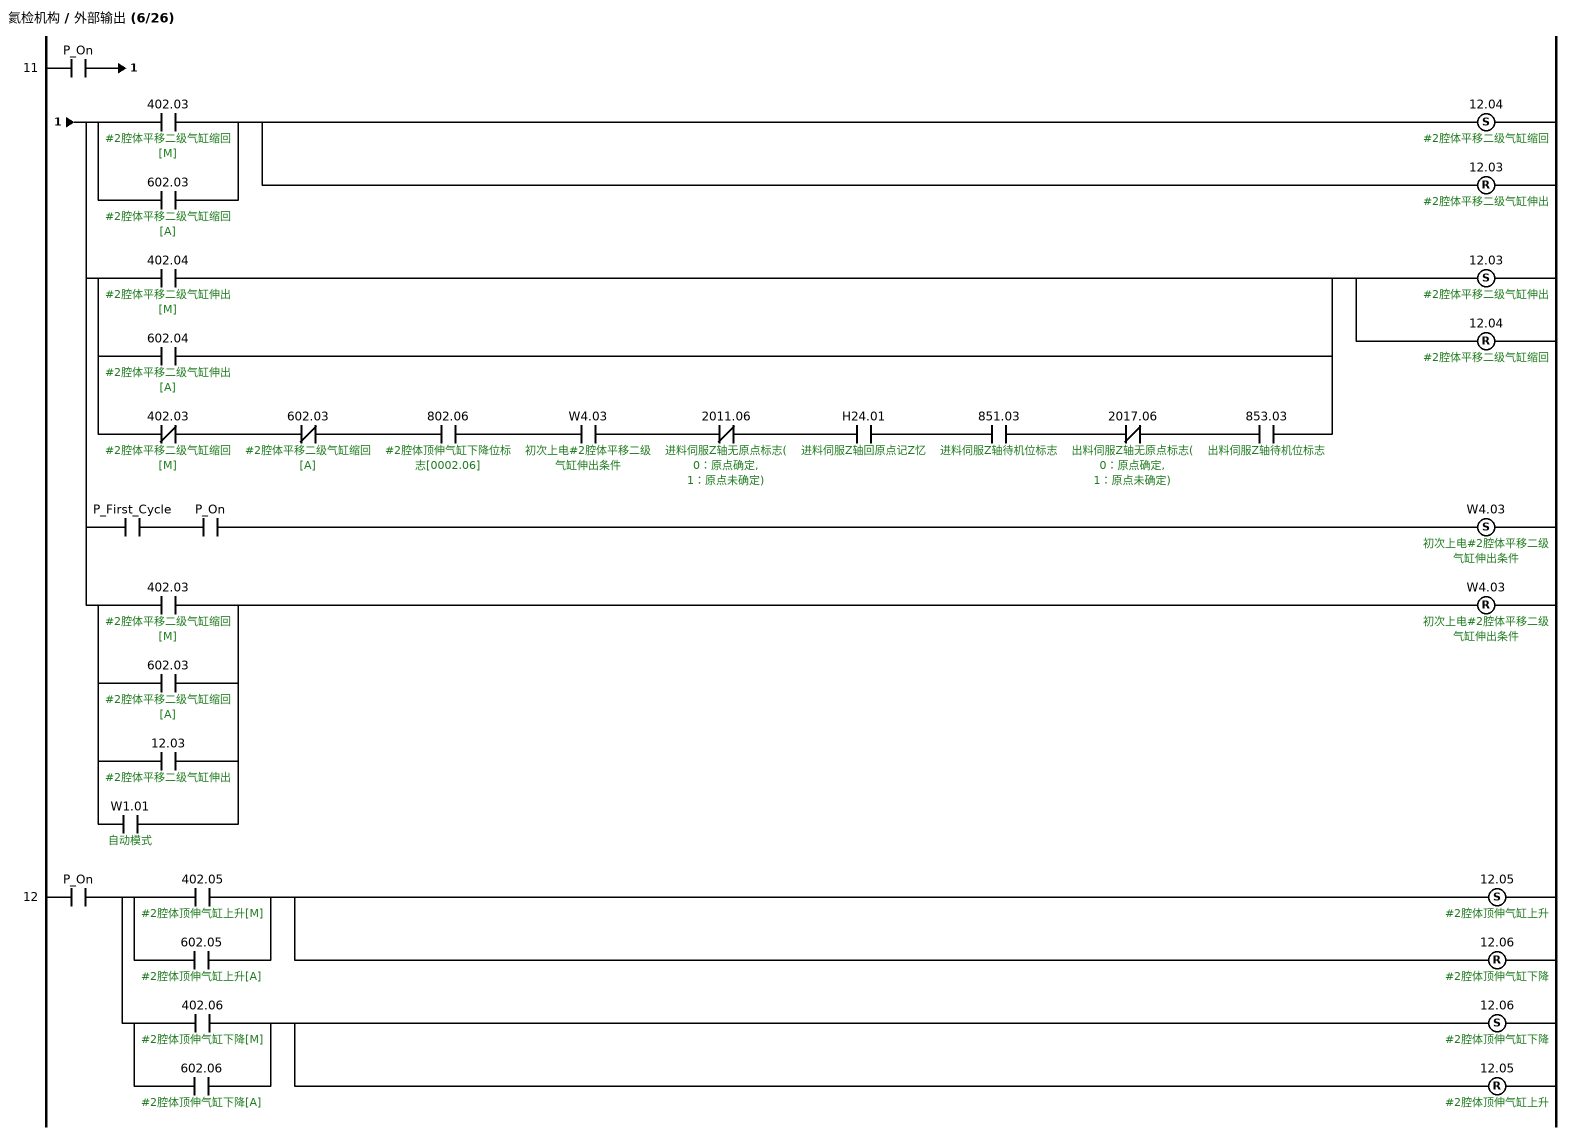
; [picture p432: 氦检机构 / 外部输出, rungs 11-12]
; rung 11
LD P_On
OUT TR0
LD 402.03  ; #2腔体平移二级气缸缩回[M]
OR 602.03  ; #2腔体平移二级气缸缩回[A]
ANDLD
SET 12.04  ; #2腔体平移二级气缸缩回
RSET 12.03  ; #2腔体平移二级气缸伸出
LD TR0
LD 402.04  ; #2腔体平移二级气缸伸出[M]
OR 602.04  ; #2腔体平移二级气缸伸出[A]
LDNOT 402.03  ; #2腔体平移二级气缸缩回[M]
ANDNOT 602.03  ; #2腔体平移二级气缸缩回[A]
AND 802.06  ; #2腔体顶伸气缸下降位标志[0002.06]
AND W4.03  ; 初次上电#2腔体平移二级气缸伸出条件
ANDNOT 2011.06  ; 进料伺服Z轴无原点标志(0：原点确定,1：原点未确定)
AND H24.01  ; 进料伺服Z轴回原点记Z忆
AND 851.03  ; 进料伺服Z轴待机位标志
ANDNOT 2017.06  ; 出料伺服Z轴无原点标志(0：原点确定,1：原点未确定)
AND 853.03  ; 出料伺服Z轴待机位标志
ORLD
ANDLD
SET 12.03  ; #2腔体平移二级气缸伸出
RSET 12.04  ; #2腔体平移二级气缸缩回
LD TR0
AND P_First_Cycle
AND P_On
SET W4.03  ; 初次上电#2腔体平移二级气缸伸出条件
LD TR0
LD 402.03  ; #2腔体平移二级气缸缩回[M]
OR 602.03  ; #2腔体平移二级气缸缩回[A]
OR 12.03  ; #2腔体平移二级气缸伸出
OR W1.01  ; 自动模式
ANDLD
RSET W4.03  ; 初次上电#2腔体平移二级气缸伸出条件
; rung 12
LD P_On
OUT TR0
LD 402.05  ; #2腔体顶伸气缸上升[M]
OR 602.05  ; #2腔体顶伸气缸上升[A]
ANDLD
SET 12.05  ; #2腔体顶伸气缸上升
RSET 12.06  ; #2腔体顶伸气缸下降
LD TR0
LD 402.06  ; #2腔体顶伸气缸下降[M]
OR 602.06  ; #2腔体顶伸气缸下降[A]
ANDLD
SET 12.06  ; #2腔体顶伸气缸下降
RSET 12.05  ; #2腔体顶伸气缸上升

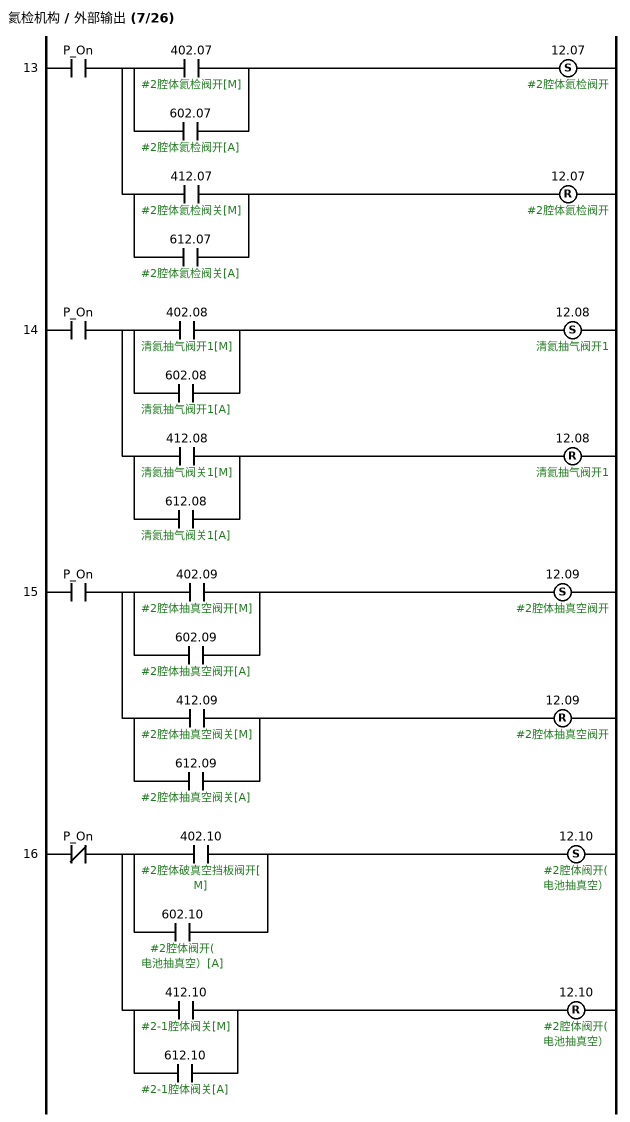
; rung 13
LD P_On
OUT TR0
LD 402.07  ; #2腔体氦检阀开[M]
OR 602.07  ; #2腔体氦检阀开[A]
ANDLD
SET 12.07  ; #2腔体氦检阀开
LD TR0
LD 412.07  ; #2腔体氦检阀关[M]
OR 612.07  ; #2腔体氦检阀关[A]
ANDLD
RSET 12.07  ; #2腔体氦检阀开
; rung 14
LD P_On
OUT TR0
LD 402.08  ; 清氦抽气阀开1[M]
OR 602.08  ; 清氦抽气阀开1[A]
ANDLD
SET 12.08  ; 清氦抽气阀开1
LD TR0
LD 412.08  ; 清氦抽气阀关1[M]
OR 612.08  ; 清氦抽气阀关1[A]
ANDLD
RSET 12.08  ; 清氦抽气阀开1
; rung 15
LD P_On
OUT TR0
LD 402.09  ; #2腔体抽真空阀开[M]
OR 602.09  ; #2腔体抽真空阀开[A]
ANDLD
SET 12.09  ; #2腔体抽真空阀开
LD TR0
LD 412.09  ; #2腔体抽真空阀关[M]
OR 612.09  ; #2腔体抽真空阀关[A]
ANDLD
RSET 12.09  ; #2腔体抽真空阀开
; rung 16
LDNOT P_On
OUT TR0
LD 402.10  ; #2腔体破真空挡板阀开[M]
OR 602.10  ; #2腔体阀开(电池抽真空）[A]
ANDLD
SET 12.10  ; #2腔体阀开(电池抽真空）
LD TR0
LD 412.10  ; #2-1腔体阀关[M]
OR 612.10  ; #2-1腔体阀关[A]
ANDLD
RSET 12.10  ; #2腔体阀开(电池抽真空）

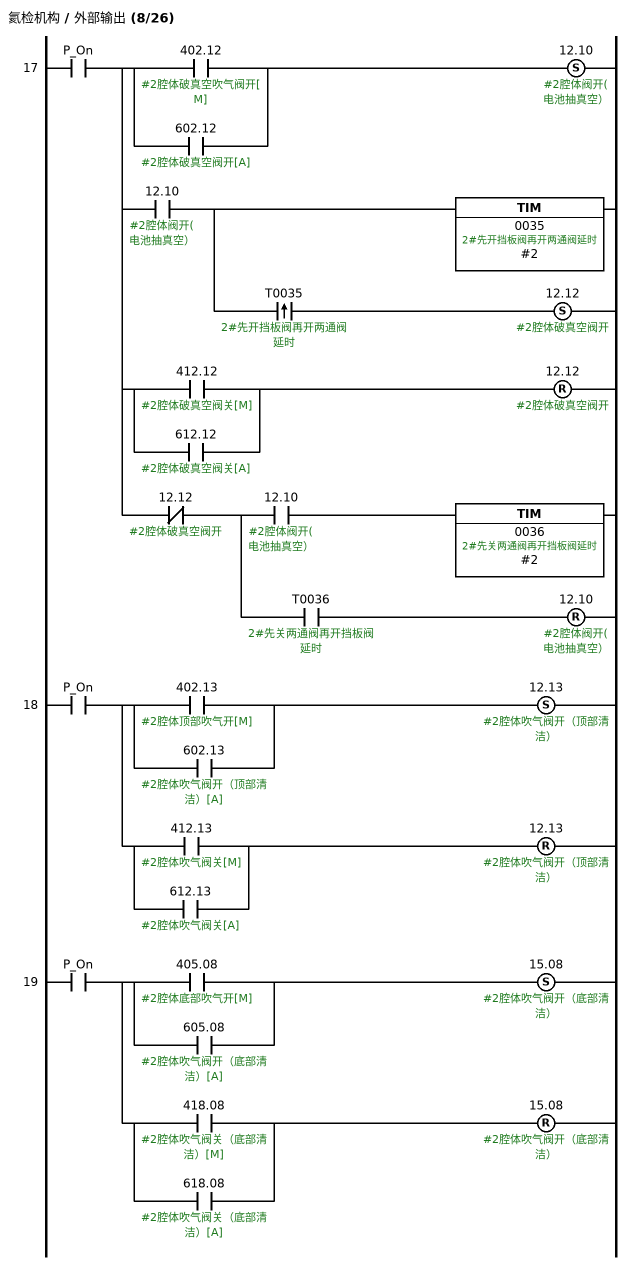
; rung 17
LD P_On
OUT TR0
LD 402.12  ; #2腔体破真空吹气阀开[M]
OR 602.12  ; #2腔体破真空阀开[A]
ANDLD
SET 12.10  ; #2腔体阀开(电池抽真空）
LD TR0
AND 12.10  ; #2腔体阀开(电池抽真空）
TIM 0035 #2  ; 2#先开挡板阀再开两通阀延时
@AND T0035  ; 2#先开挡板阀再开两通阀延时
SET 12.12  ; #2腔体破真空阀开
LD TR0
LD 412.12  ; #2腔体破真空阀关[M]
OR 612.12  ; #2腔体破真空阀关[A]
ANDLD
RSET 12.12  ; #2腔体破真空阀开
LD TR0
ANDNOT 12.12  ; #2腔体破真空阀开
OUT TR0
AND 12.10  ; #2腔体阀开(电池抽真空）
TIM 0036 #2  ; 2#先关两通阀再开挡板阀延时
LD TR0
AND T0036  ; 2#先关两通阀再开挡板阀延时
RSET 12.10  ; #2腔体阀开(电池抽真空）
; rung 18
LD P_On
OUT TR0
LD 402.13  ; #2腔体顶部吹气开[M]
OR 602.13  ; #2腔体吹气阀开（顶部清洁）[A]
ANDLD
SET 12.13  ; #2腔体吹气阀开（顶部清洁）
LD TR0
LD 412.13  ; #2腔体吹气阀关[M]
OR 612.13  ; #2腔体吹气阀关[A]
ANDLD
RSET 12.13  ; #2腔体吹气阀开（顶部清洁）
; rung 19
LD P_On
OUT TR0
LD 405.08  ; #2腔体底部吹气开[M]
OR 605.08  ; #2腔体吹气阀开（底部清洁）[A]
ANDLD
SET 15.08  ; #2腔体吹气阀开（底部清洁）
LD TR0
LD 418.08  ; #2腔体吹气阀关（底部清洁）[M]
OR 618.08  ; #2腔体吹气阀关（底部清洁）[A]
ANDLD
RSET 15.08  ; #2腔体吹气阀开（底部清洁）

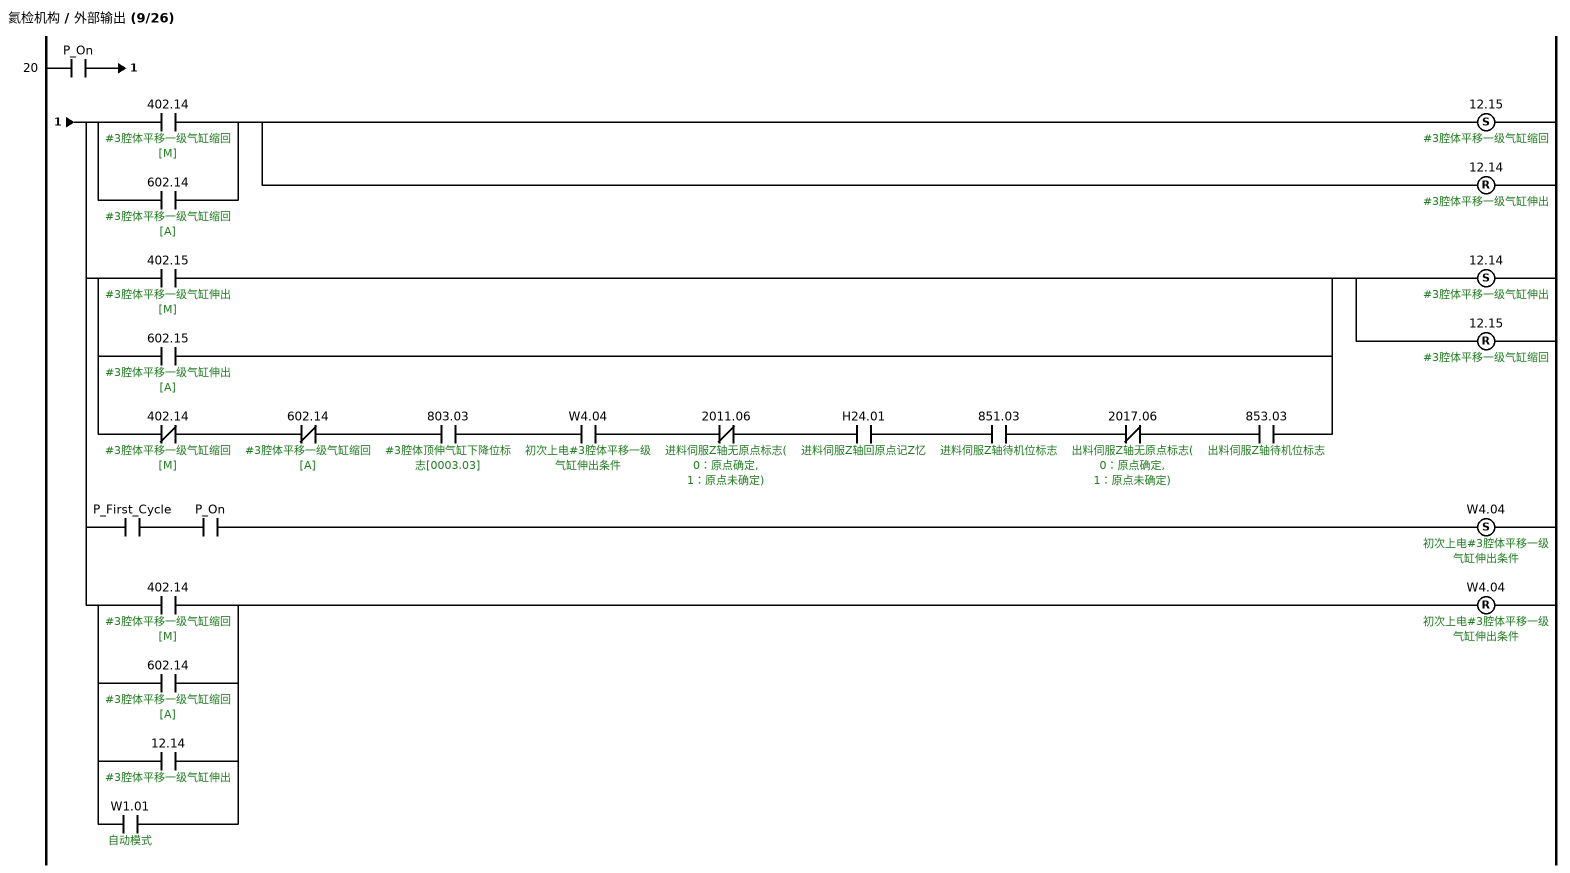
; rung 20
LD P_On
OUT TR0
LD 402.14  ; #3腔体平移一级气缸缩回[M]
OR 602.14  ; #3腔体平移一级气缸缩回[A]
ANDLD
SET 12.15  ; #3腔体平移一级气缸缩回
RSET 12.14  ; #3腔体平移一级气缸伸出
LD TR0
LD 402.15  ; #3腔体平移一级气缸伸出[M]
OR 602.15  ; #3腔体平移一级气缸伸出[A]
LDNOT 402.14  ; #3腔体平移一级气缸缩回[M]
ANDNOT 602.14  ; #3腔体平移一级气缸缩回[A]
AND 803.03  ; #3腔体顶伸气缸下降位标志[0003.03]
AND W4.04  ; 初次上电#3腔体平移一级气缸伸出条件
ANDNOT 2011.06  ; 进料伺服Z轴无原点标志(0：原点确定,1：原点未确定)
AND H24.01  ; 进料伺服Z轴回原点记Z忆
AND 851.03  ; 进料伺服Z轴待机位标志
ANDNOT 2017.06  ; 出料伺服Z轴无原点标志(0：原点确定,1：原点未确定)
AND 853.03  ; 出料伺服Z轴待机位标志
ORLD
ANDLD
SET 12.14  ; #3腔体平移一级气缸伸出
RSET 12.15  ; #3腔体平移一级气缸缩回
LD TR0
AND P_First_Cycle
AND P_On
SET W4.04  ; 初次上电#3腔体平移一级气缸伸出条件
LD TR0
LD 402.14  ; #3腔体平移一级气缸缩回[M]
OR 602.14  ; #3腔体平移一级气缸缩回[A]
OR 12.14  ; #3腔体平移一级气缸伸出
OR W1.01  ; 自动模式
ANDLD
RSET W4.04  ; 初次上电#3腔体平移一级气缸伸出条件

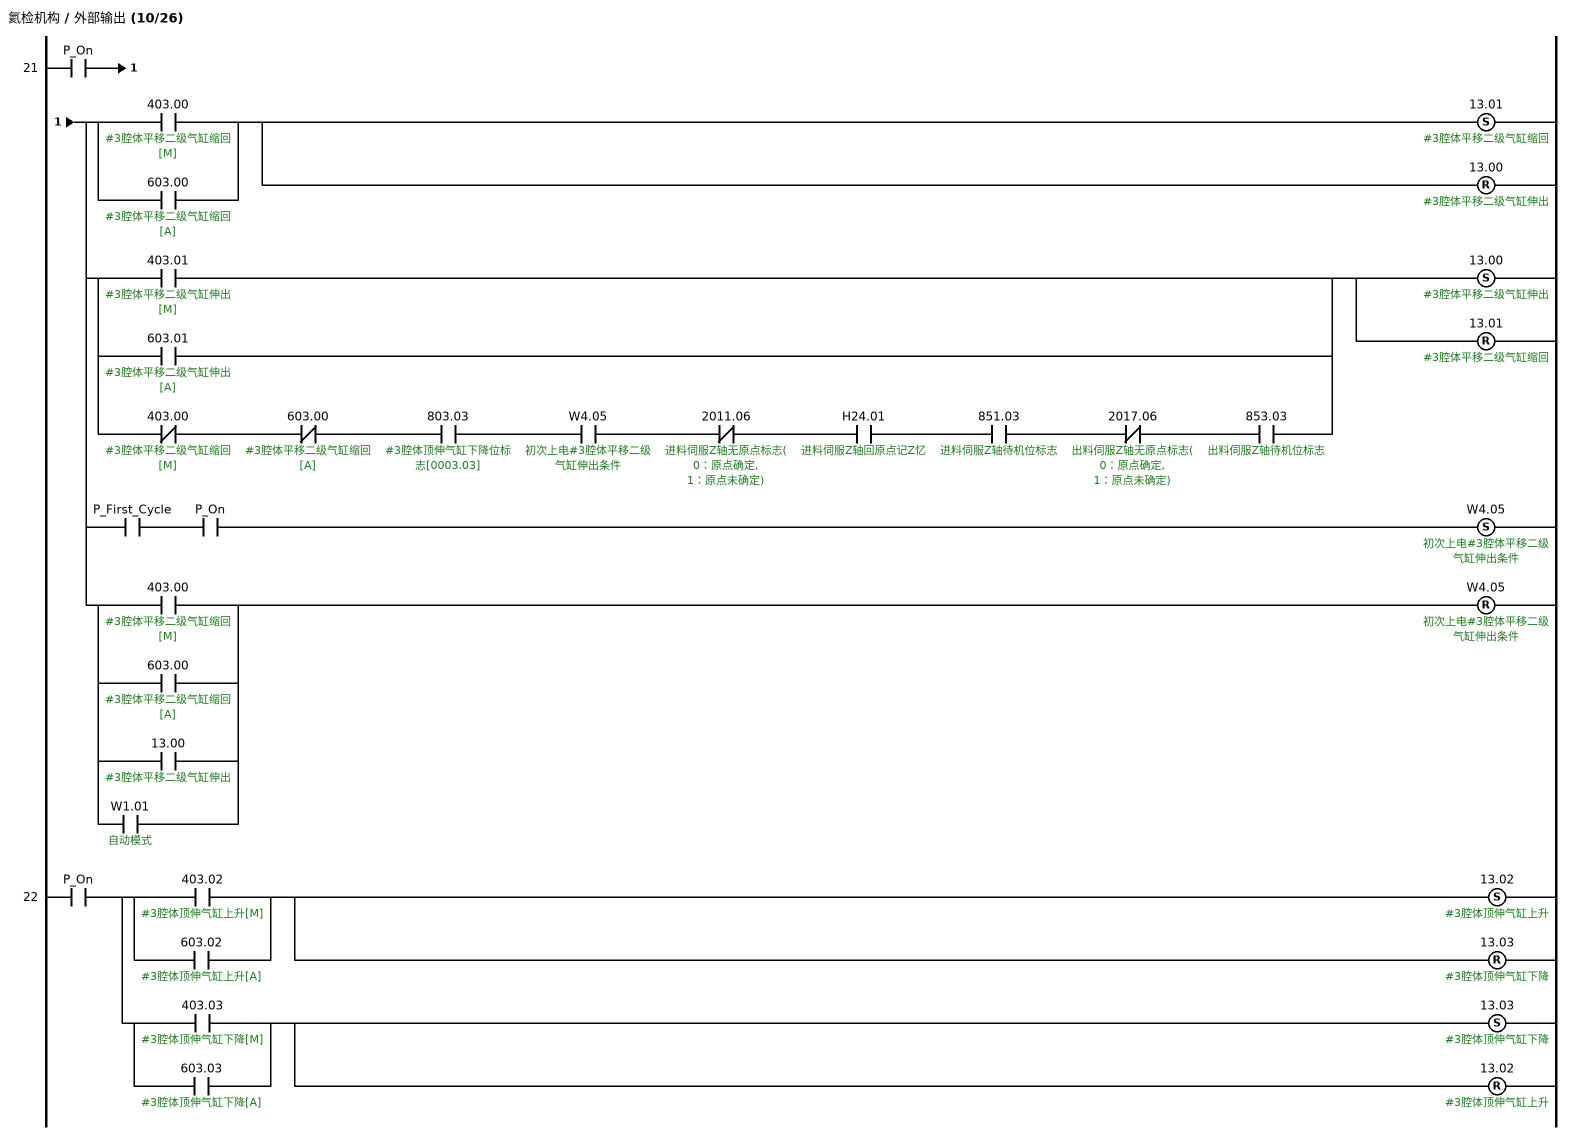
; rung 21
LD P_On
OUT TR0
LD 403.00  ; #3腔体平移二级气缸缩回[M]
OR 603.00  ; #3腔体平移二级气缸缩回[A]
ANDLD
SET 13.01  ; #3腔体平移二级气缸缩回
RSET 13.00  ; #3腔体平移二级气缸伸出
LD TR0
LD 403.01  ; #3腔体平移二级气缸伸出[M]
OR 603.01  ; #3腔体平移二级气缸伸出[A]
LDNOT 403.00  ; #3腔体平移二级气缸缩回[M]
ANDNOT 603.00  ; #3腔体平移二级气缸缩回[A]
AND 803.03  ; #3腔体顶伸气缸下降位标志[0003.03]
AND W4.05  ; 初次上电#3腔体平移二级气缸伸出条件
ANDNOT 2011.06  ; 进料伺服Z轴无原点标志(0：原点确定,1：原点未确定)
AND H24.01  ; 进料伺服Z轴回原点记Z忆
AND 851.03  ; 进料伺服Z轴待机位标志
ANDNOT 2017.06  ; 出料伺服Z轴无原点标志(0：原点确定,1：原点未确定)
AND 853.03  ; 出料伺服Z轴待机位标志
ORLD
ANDLD
SET 13.00  ; #3腔体平移二级气缸伸出
RSET 13.01  ; #3腔体平移二级气缸缩回
LD TR0
AND P_First_Cycle
AND P_On
SET W4.05  ; 初次上电#3腔体平移二级气缸伸出条件
LD TR0
LD 403.00  ; #3腔体平移二级气缸缩回[M]
OR 603.00  ; #3腔体平移二级气缸缩回[A]
OR 13.00  ; #3腔体平移二级气缸伸出
OR W1.01  ; 自动模式
ANDLD
RSET W4.05  ; 初次上电#3腔体平移二级气缸伸出条件
; rung 22
LD P_On
OUT TR0
LD 403.02  ; #3腔体顶伸气缸上升[M]
OR 603.02  ; #3腔体顶伸气缸上升[A]
ANDLD
SET 13.02  ; #3腔体顶伸气缸上升
RSET 13.03  ; #3腔体顶伸气缸下降
LD TR0
LD 403.03  ; #3腔体顶伸气缸下降[M]
OR 603.03  ; #3腔体顶伸气缸下降[A]
ANDLD
SET 13.03  ; #3腔体顶伸气缸下降
RSET 13.02  ; #3腔体顶伸气缸上升

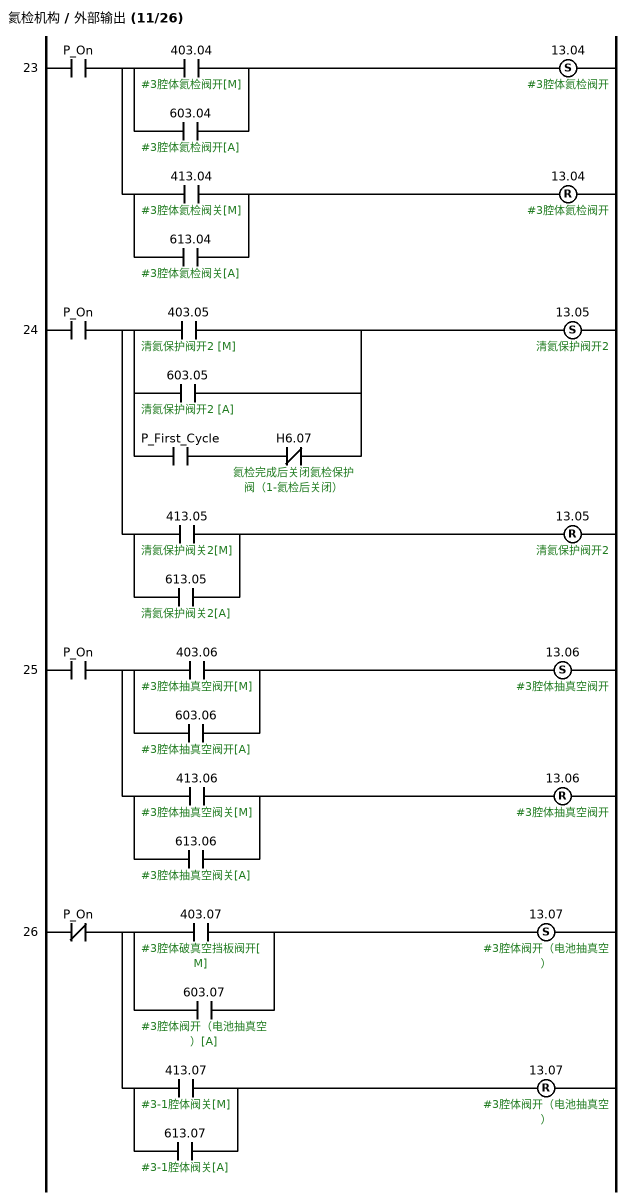
; rung 23
LD P_On
OUT TR0
LD 403.04  ; #3腔体氦检阀开[M]
OR 603.04  ; #3腔体氦检阀开[A]
ANDLD
SET 13.04  ; #3腔体氦检阀开
LD TR0
LD 413.04  ; #3腔体氦检阀关[M]
OR 613.04  ; #3腔体氦检阀关[A]
ANDLD
RSET 13.04  ; #3腔体氦检阀开
; rung 24
LD P_On
OUT TR0
LD 403.05  ; 清氦保护阀开2 [M]
OR 603.05  ; 清氦保护阀开2 [A]
LD P_First_Cycle  // 保证氦检仪开启时能将管路抽成真空状态
ANDNOT H6.07  ; 氦检完成后关闭氦检保护阀（1-氦检后关闭）
ORLD
ANDLD
SET 13.05  ; 清氦保护阀开2
LD TR0
LD 413.05  ; 清氦保护阀关2[M]
OR 613.05  ; 清氦保护阀关2[A]
ANDLD
RSET 13.05  ; 清氦保护阀开2
; rung 25
LD P_On
OUT TR0
LD 403.06  ; #3腔体抽真空阀开[M]
OR 603.06  ; #3腔体抽真空阀开[A]
ANDLD
SET 13.06  ; #3腔体抽真空阀开
LD TR0
LD 413.06  ; #3腔体抽真空阀关[M]
OR 613.06  ; #3腔体抽真空阀关[A]
ANDLD
RSET 13.06  ; #3腔体抽真空阀开
; rung 26
LDNOT P_On
OUT TR0
LD 403.07  ; #3腔体破真空挡板阀开[M]
OR 603.07  ; #3腔体阀开（电池抽真空）[A]
ANDLD
SET 13.07  ; #3腔体阀开（电池抽真空）
LD TR0
LD 413.07  ; #3-1腔体阀关[M]
OR 613.07  ; #3-1腔体阀关[A]
ANDLD
RSET 13.07  ; #3腔体阀开（电池抽真空）

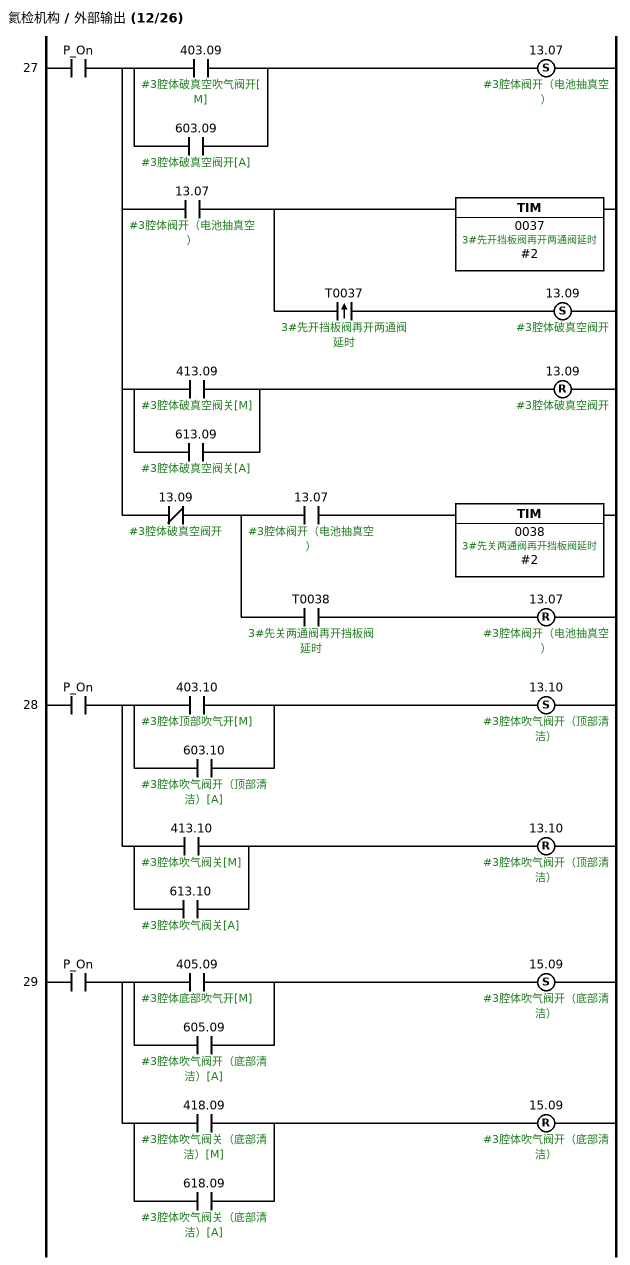
; rung 27
LD P_On
OUT TR0
LD 403.09  ; #3腔体破真空吹气阀开[M]
OR 603.09  ; #3腔体破真空阀开[A]
ANDLD
SET 13.07  ; #3腔体阀开（电池抽真空）
LD TR0
AND 13.07  ; #3腔体阀开（电池抽真空）
TIM 0037 #2  ; 3#先开挡板阀再开两通阀延时
@AND T0037  ; 3#先开挡板阀再开两通阀延时
SET 13.09  ; #3腔体破真空阀开
LD TR0
LD 413.09  ; #3腔体破真空阀关[M]
OR 613.09  ; #3腔体破真空阀关[A]
ANDLD
RSET 13.09  ; #3腔体破真空阀开
LD TR0
ANDNOT 13.09  ; #3腔体破真空阀开
OUT TR0
AND 13.07  ; #3腔体阀开（电池抽真空）
TIM 0038 #2  ; 3#先关两通阀再开挡板阀延时
LD TR0
AND T0038  ; 3#先关两通阀再开挡板阀延时
RSET 13.07  ; #3腔体阀开（电池抽真空）
; rung 28
LD P_On
OUT TR0
LD 403.10  ; #3腔体顶部吹气开[M]
OR 603.10  ; #3腔体吹气阀开（顶部清洁）[A]
ANDLD
SET 13.10  ; #3腔体吹气阀开（顶部清洁）
LD TR0
LD 413.10  ; #3腔体吹气阀关[M]
OR 613.10  ; #3腔体吹气阀关[A]
ANDLD
RSET 13.10  ; #3腔体吹气阀开（顶部清洁）
; rung 29
LD P_On
OUT TR0
LD 405.09  ; #3腔体底部吹气开[M]
OR 605.09  ; #3腔体吹气阀开（底部清洁）[A]
ANDLD
SET 15.09  ; #3腔体吹气阀开（底部清洁）
LD TR0
LD 418.09  ; #3腔体吹气阀关（底部清洁）[M]
OR 618.09  ; #3腔体吹气阀关（底部清洁）[A]
ANDLD
RSET 15.09  ; #3腔体吹气阀开（底部清洁）

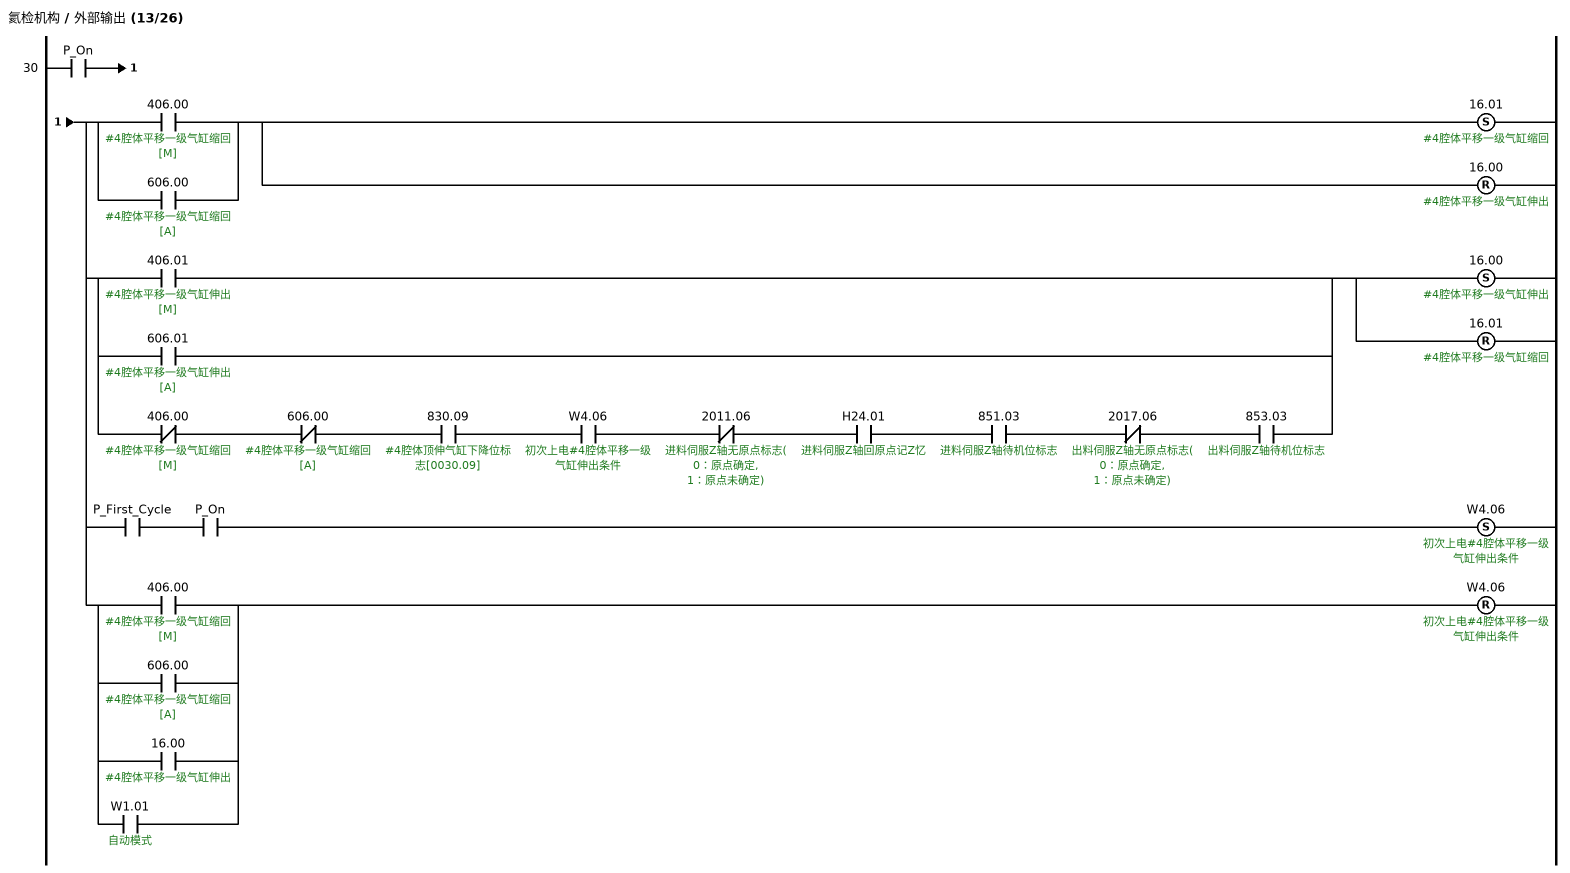
; rung 30
LD P_On
OUT TR0
LD 406.00  ; #4腔体平移一级气缸缩回[M]
OR 606.00  ; #4腔体平移一级气缸缩回[A]
ANDLD
SET 16.01  ; #4腔体平移一级气缸缩回
RSET 16.00  ; #4腔体平移一级气缸伸出
LD TR0
LD 406.01  ; #4腔体平移一级气缸伸出[M]
OR 606.01  ; #4腔体平移一级气缸伸出[A]
LDNOT 406.00  ; #4腔体平移一级气缸缩回[M]
ANDNOT 606.00  ; #4腔体平移一级气缸缩回[A]
AND 830.09  ; #4腔体顶伸气缸下降位标志[0030.09]
AND W4.06  ; 初次上电#4腔体平移一级气缸伸出条件
ANDNOT 2011.06  ; 进料伺服Z轴无原点标志(0：原点确定,1：原点未确定)
AND H24.01  ; 进料伺服Z轴回原点记Z忆
AND 851.03  ; 进料伺服Z轴待机位标志
ANDNOT 2017.06  ; 出料伺服Z轴无原点标志(0：原点确定,1：原点未确定)
AND 853.03  ; 出料伺服Z轴待机位标志
ORLD
ANDLD
SET 16.00  ; #4腔体平移一级气缸伸出
RSET 16.01  ; #4腔体平移一级气缸缩回
LD TR0
AND P_First_Cycle
AND P_On
SET W4.06  ; 初次上电#4腔体平移一级气缸伸出条件
LD TR0
LD 406.00  ; #4腔体平移一级气缸缩回[M]
OR 606.00  ; #4腔体平移一级气缸缩回[A]
OR 16.00  ; #4腔体平移一级气缸伸出
OR W1.01  ; 自动模式
ANDLD
RSET W4.06  ; 初次上电#4腔体平移一级气缸伸出条件

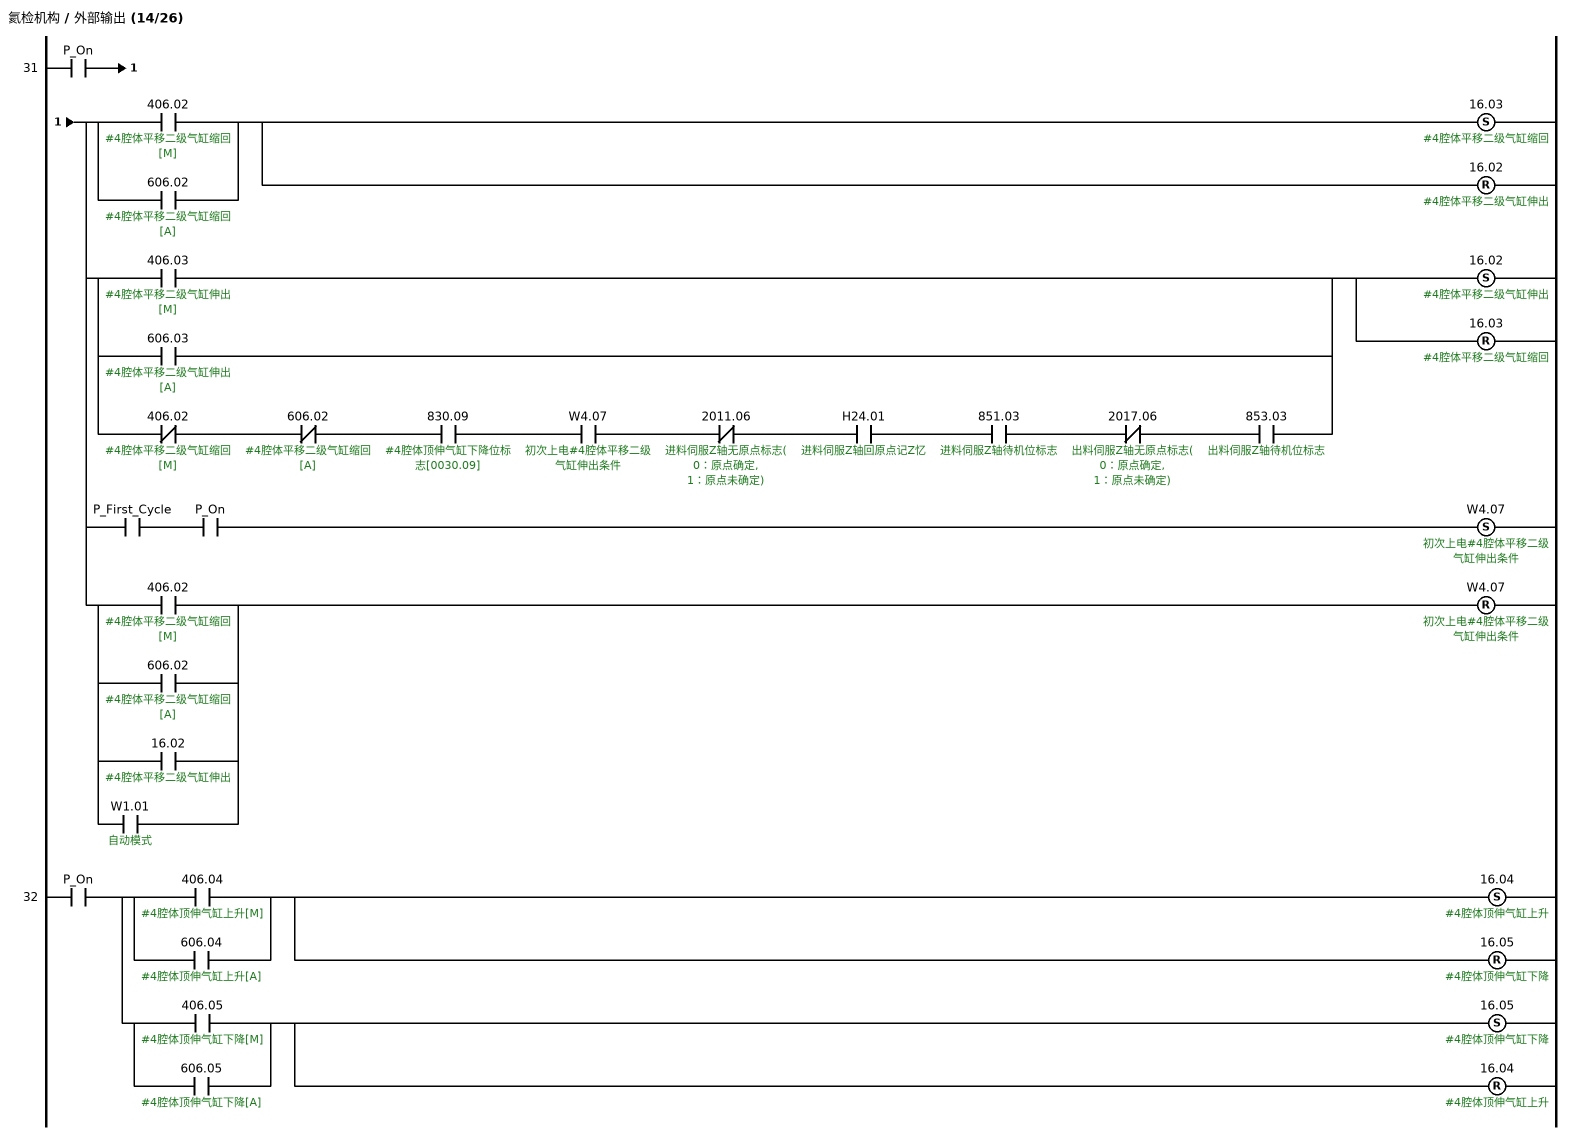
; rung 31
LD P_On
OUT TR0
LD 406.02  ; #4腔体平移二级气缸缩回[M]
OR 606.02  ; #4腔体平移二级气缸缩回[A]
ANDLD
SET 16.03  ; #4腔体平移二级气缸缩回
RSET 16.02  ; #4腔体平移二级气缸伸出
LD TR0
LD 406.03  ; #4腔体平移二级气缸伸出[M]
OR 606.03  ; #4腔体平移二级气缸伸出[A]
LDNOT 406.02  ; #4腔体平移二级气缸缩回[M]
ANDNOT 606.02  ; #4腔体平移二级气缸缩回[A]
AND 830.09  ; #4腔体顶伸气缸下降位标志[0030.09]
AND W4.07  ; 初次上电#4腔体平移二级气缸伸出条件
ANDNOT 2011.06  ; 进料伺服Z轴无原点标志(0：原点确定,1：原点未确定)
AND H24.01  ; 进料伺服Z轴回原点记Z忆
AND 851.03  ; 进料伺服Z轴待机位标志
ANDNOT 2017.06  ; 出料伺服Z轴无原点标志(0：原点确定,1：原点未确定)
AND 853.03  ; 出料伺服Z轴待机位标志
ORLD
ANDLD
SET 16.02  ; #4腔体平移二级气缸伸出
RSET 16.03  ; #4腔体平移二级气缸缩回
LD TR0
AND P_First_Cycle
AND P_On
SET W4.07  ; 初次上电#4腔体平移二级气缸伸出条件
LD TR0
LD 406.02  ; #4腔体平移二级气缸缩回[M]
OR 606.02  ; #4腔体平移二级气缸缩回[A]
OR 16.02  ; #4腔体平移二级气缸伸出
OR W1.01  ; 自动模式
ANDLD
RSET W4.07  ; 初次上电#4腔体平移二级气缸伸出条件
; rung 32
LD P_On
OUT TR0
LD 406.04  ; #4腔体顶伸气缸上升[M]
OR 606.04  ; #4腔体顶伸气缸上升[A]
ANDLD
SET 16.04  ; #4腔体顶伸气缸上升
RSET 16.05  ; #4腔体顶伸气缸下降
LD TR0
LD 406.05  ; #4腔体顶伸气缸下降[M]
OR 606.05  ; #4腔体顶伸气缸下降[A]
ANDLD
SET 16.05  ; #4腔体顶伸气缸下降
RSET 16.04  ; #4腔体顶伸气缸上升

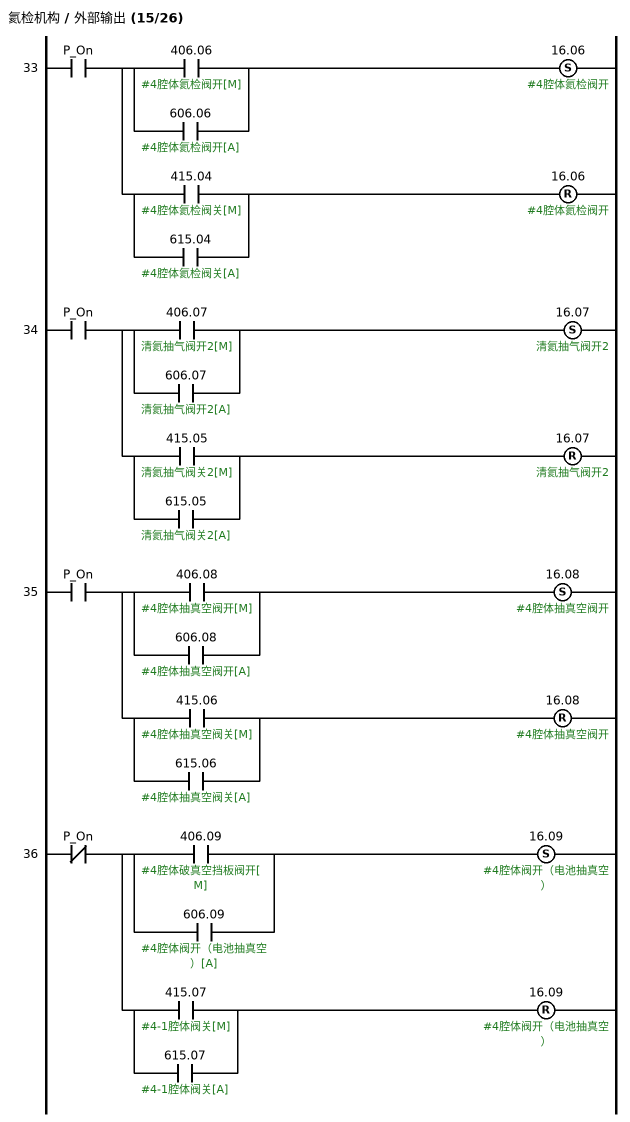
; rung 33
LD P_On
OUT TR0
LD 406.06  ; #4腔体氦检阀开[M]
OR 606.06  ; #4腔体氦检阀开[A]
ANDLD
SET 16.06  ; #4腔体氦检阀开
LD TR0
LD 415.04  ; #4腔体氦检阀关[M]
OR 615.04  ; #4腔体氦检阀关[A]
ANDLD
RSET 16.06  ; #4腔体氦检阀开
; rung 34
LD P_On
OUT TR0
LD 406.07  ; 清氦抽气阀开2[M]
OR 606.07  ; 清氦抽气阀开2[A]
ANDLD
SET 16.07  ; 清氦抽气阀开2
LD TR0
LD 415.05  ; 清氦抽气阀关2[M]
OR 615.05  ; 清氦抽气阀关2[A]
ANDLD
RSET 16.07  ; 清氦抽气阀开2
; rung 35
LD P_On
OUT TR0
LD 406.08  ; #4腔体抽真空阀开[M]
OR 606.08  ; #4腔体抽真空阀开[A]
ANDLD
SET 16.08  ; #4腔体抽真空阀开
LD TR0
LD 415.06  ; #4腔体抽真空阀关[M]
OR 615.06  ; #4腔体抽真空阀关[A]
ANDLD
RSET 16.08  ; #4腔体抽真空阀开
; rung 36
LDNOT P_On
OUT TR0
LD 406.09  ; #4腔体破真空挡板阀开[M]
OR 606.09  ; #4腔体阀开（电池抽真空）[A]
ANDLD
SET 16.09  ; #4腔体阀开（电池抽真空）
LD TR0
LD 415.07  ; #4-1腔体阀关[M]
OR 615.07  ; #4-1腔体阀关[A]
ANDLD
RSET 16.09  ; #4腔体阀开（电池抽真空）

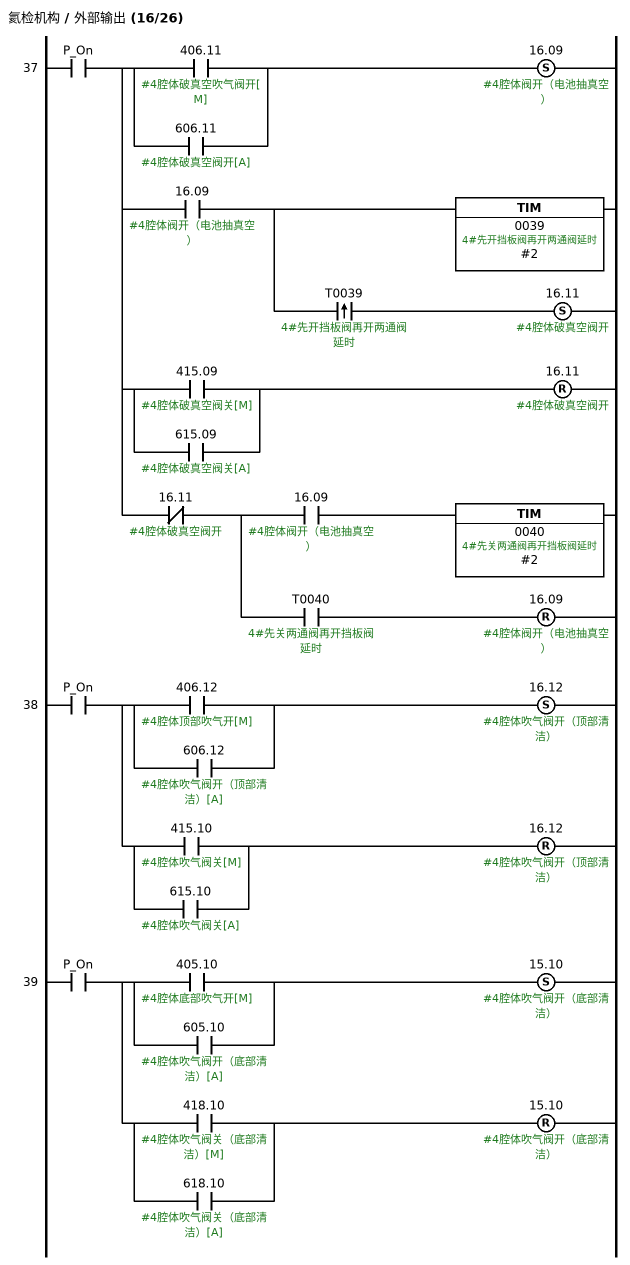
; rung 37
LD P_On
OUT TR0
LD 406.11  ; #4腔体破真空吹气阀开[M]
OR 606.11  ; #4腔体破真空阀开[A]
ANDLD
SET 16.09  ; #4腔体阀开（电池抽真空）
LD TR0
AND 16.09  ; #4腔体阀开（电池抽真空）
TIM 0039 #2  ; 4#先开挡板阀再开两通阀延时
@AND T0039  ; 4#先开挡板阀再开两通阀延时
SET 16.11  ; #4腔体破真空阀开
LD TR0
LD 415.09  ; #4腔体破真空阀关[M]
OR 615.09  ; #4腔体破真空阀关[A]
ANDLD
RSET 16.11  ; #4腔体破真空阀开
LD TR0
ANDNOT 16.11  ; #4腔体破真空阀开
OUT TR0
AND 16.09  ; #4腔体阀开（电池抽真空）
TIM 0040 #2  ; 4#先关两通阀再开挡板阀延时
LD TR0
AND T0040  ; 4#先关两通阀再开挡板阀延时
RSET 16.09  ; #4腔体阀开（电池抽真空）
; rung 38
LD P_On
OUT TR0
LD 406.12  ; #4腔体顶部吹气开[M]
OR 606.12  ; #4腔体吹气阀开（顶部清洁）[A]
ANDLD
SET 16.12  ; #4腔体吹气阀开（顶部清洁）
LD TR0
LD 415.10  ; #4腔体吹气阀关[M]
OR 615.10  ; #4腔体吹气阀关[A]
ANDLD
RSET 16.12  ; #4腔体吹气阀开（顶部清洁）
; rung 39
LD P_On
OUT TR0
LD 405.10  ; #4腔体底部吹气开[M]
OR 605.10  ; #4腔体吹气阀开（底部清洁）[A]
ANDLD
SET 15.10  ; #4腔体吹气阀开（底部清洁）
LD TR0
LD 418.10  ; #4腔体吹气阀关（底部清洁）[M]
OR 618.10  ; #4腔体吹气阀关（底部清洁）[A]
ANDLD
RSET 15.10  ; #4腔体吹气阀开（底部清洁）

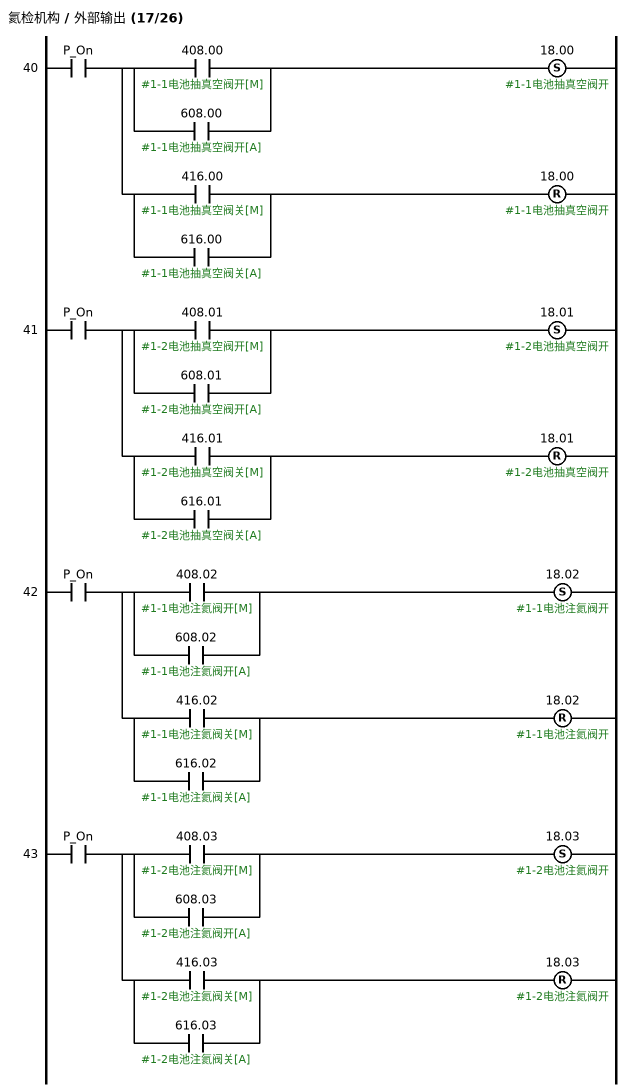
; rung 40
LD P_On
OUT TR0
LD 408.00  ; #1-1电池抽真空阀开[M]
OR 608.00  ; #1-1电池抽真空阀开[A]
ANDLD
SET 18.00  ; #1-1电池抽真空阀开
LD TR0
LD 416.00  ; #1-1电池抽真空阀关[M]
OR 616.00  ; #1-1电池抽真空阀关[A]
ANDLD
RSET 18.00  ; #1-1电池抽真空阀开
; rung 41
LD P_On
OUT TR0
LD 408.01  ; #1-2电池抽真空阀开[M]
OR 608.01  ; #1-2电池抽真空阀开[A]
ANDLD
SET 18.01  ; #1-2电池抽真空阀开
LD TR0
LD 416.01  ; #1-2电池抽真空阀关[M]
OR 616.01  ; #1-2电池抽真空阀关[A]
ANDLD
RSET 18.01  ; #1-2电池抽真空阀开
; rung 42
LD P_On
OUT TR0
LD 408.02  ; #1-1电池注氦阀开[M]
OR 608.02  ; #1-1电池注氦阀开[A]
ANDLD
SET 18.02  ; #1-1电池注氦阀开
LD TR0
LD 416.02  ; #1-1电池注氦阀关[M]
OR 616.02  ; #1-1电池注氦阀关[A]
ANDLD
RSET 18.02  ; #1-1电池注氦阀开
; rung 43
LD P_On
OUT TR0
LD 408.03  ; #1-2电池注氦阀开[M]
OR 608.03  ; #1-2电池注氦阀开[A]
ANDLD
SET 18.03  ; #1-2电池注氦阀开
LD TR0
LD 416.03  ; #1-2电池注氦阀关[M]
OR 616.03  ; #1-2电池注氦阀关[A]
ANDLD
RSET 18.03  ; #1-2电池注氦阀开

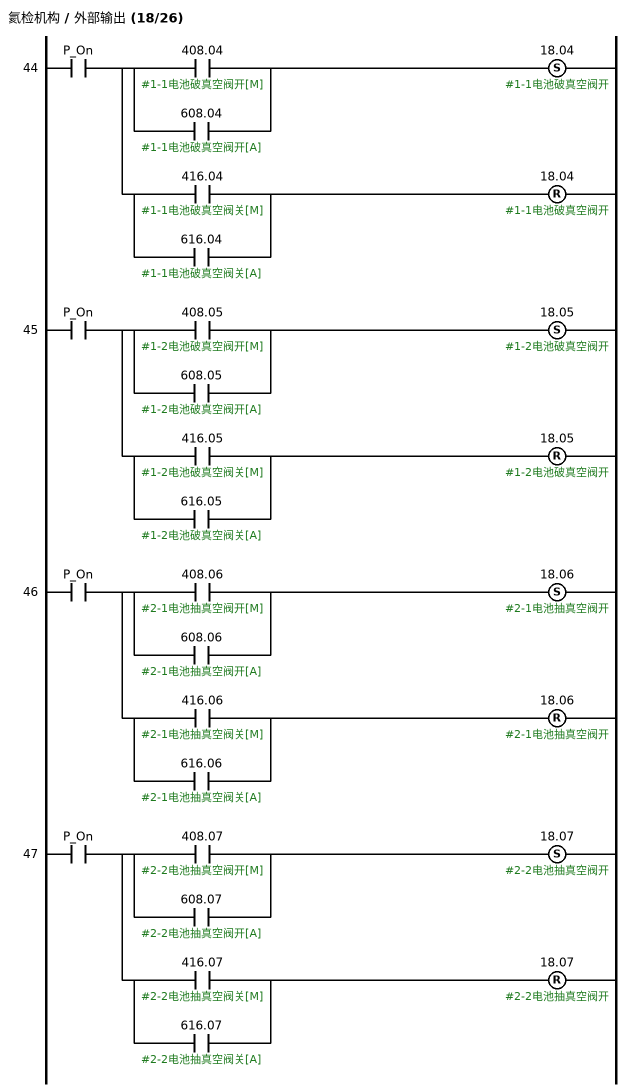
; rung 44
LD P_On
OUT TR0
LD 408.04  ; #1-1电池破真空阀开[M]
OR 608.04  ; #1-1电池破真空阀开[A]
ANDLD
SET 18.04  ; #1-1电池破真空阀开
LD TR0
LD 416.04  ; #1-1电池破真空阀关[M]
OR 616.04  ; #1-1电池破真空阀关[A]
ANDLD
RSET 18.04  ; #1-1电池破真空阀开
; rung 45
LD P_On
OUT TR0
LD 408.05  ; #1-2电池破真空阀开[M]
OR 608.05  ; #1-2电池破真空阀开[A]
ANDLD
SET 18.05  ; #1-2电池破真空阀开
LD TR0
LD 416.05  ; #1-2电池破真空阀关[M]
OR 616.05  ; #1-2电池破真空阀关[A]
ANDLD
RSET 18.05  ; #1-2电池破真空阀开
; rung 46
LD P_On
OUT TR0
LD 408.06  ; #2-1电池抽真空阀开[M]
OR 608.06  ; #2-1电池抽真空阀开[A]
ANDLD
SET 18.06  ; #2-1电池抽真空阀开
LD TR0
LD 416.06  ; #2-1电池抽真空阀关[M]
OR 616.06  ; #2-1电池抽真空阀关[A]
ANDLD
RSET 18.06  ; #2-1电池抽真空阀开
; rung 47
LD P_On
OUT TR0
LD 408.07  ; #2-2电池抽真空阀开[M]
OR 608.07  ; #2-2电池抽真空阀开[A]
ANDLD
SET 18.07  ; #2-2电池抽真空阀开
LD TR0
LD 416.07  ; #2-2电池抽真空阀关[M]
OR 616.07  ; #2-2电池抽真空阀关[A]
ANDLD
RSET 18.07  ; #2-2电池抽真空阀开

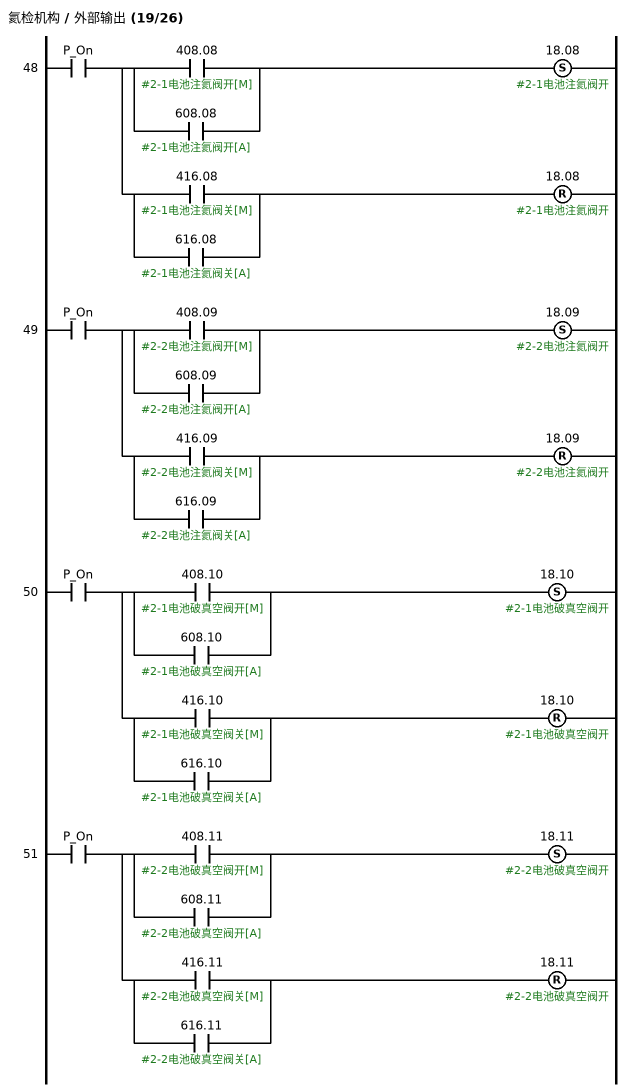
; rung 48
LD P_On
OUT TR0
LD 408.08  ; #2-1电池注氦阀开[M]
OR 608.08  ; #2-1电池注氦阀开[A]
ANDLD
SET 18.08  ; #2-1电池注氦阀开
LD TR0
LD 416.08  ; #2-1电池注氦阀关[M]
OR 616.08  ; #2-1电池注氦阀关[A]
ANDLD
RSET 18.08  ; #2-1电池注氦阀开
; rung 49
LD P_On
OUT TR0
LD 408.09  ; #2-2电池注氦阀开[M]
OR 608.09  ; #2-2电池注氦阀开[A]
ANDLD
SET 18.09  ; #2-2电池注氦阀开
LD TR0
LD 416.09  ; #2-2电池注氦阀关[M]
OR 616.09  ; #2-2电池注氦阀关[A]
ANDLD
RSET 18.09  ; #2-2电池注氦阀开
; rung 50
LD P_On
OUT TR0
LD 408.10  ; #2-1电池破真空阀开[M]
OR 608.10  ; #2-1电池破真空阀开[A]
ANDLD
SET 18.10  ; #2-1电池破真空阀开
LD TR0
LD 416.10  ; #2-1电池破真空阀关[M]
OR 616.10  ; #2-1电池破真空阀关[A]
ANDLD
RSET 18.10  ; #2-1电池破真空阀开
; rung 51
LD P_On
OUT TR0
LD 408.11  ; #2-2电池破真空阀开[M]
OR 608.11  ; #2-2电池破真空阀开[A]
ANDLD
SET 18.11  ; #2-2电池破真空阀开
LD TR0
LD 416.11  ; #2-2电池破真空阀关[M]
OR 616.11  ; #2-2电池破真空阀关[A]
ANDLD
RSET 18.11  ; #2-2电池破真空阀开

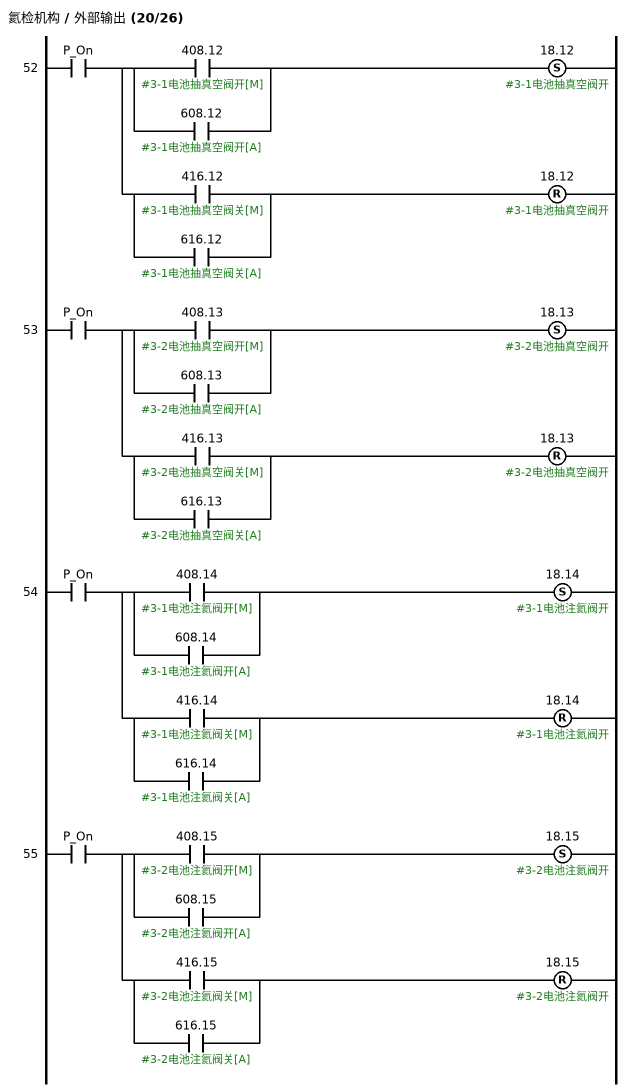
; rung 52
LD P_On
OUT TR0
LD 408.12  ; #3-1电池抽真空阀开[M]
OR 608.12  ; #3-1电池抽真空阀开[A]
ANDLD
SET 18.12  ; #3-1电池抽真空阀开
LD TR0
LD 416.12  ; #3-1电池抽真空阀关[M]
OR 616.12  ; #3-1电池抽真空阀关[A]
ANDLD
RSET 18.12  ; #3-1电池抽真空阀开
; rung 53
LD P_On
OUT TR0
LD 408.13  ; #3-2电池抽真空阀开[M]
OR 608.13  ; #3-2电池抽真空阀开[A]
ANDLD
SET 18.13  ; #3-2电池抽真空阀开
LD TR0
LD 416.13  ; #3-2电池抽真空阀关[M]
OR 616.13  ; #3-2电池抽真空阀关[A]
ANDLD
RSET 18.13  ; #3-2电池抽真空阀开
; rung 54
LD P_On
OUT TR0
LD 408.14  ; #3-1电池注氦阀开[M]
OR 608.14  ; #3-1电池注氦阀开[A]
ANDLD
SET 18.14  ; #3-1电池注氦阀开
LD TR0
LD 416.14  ; #3-1电池注氦阀关[M]
OR 616.14  ; #3-1电池注氦阀关[A]
ANDLD
RSET 18.14  ; #3-1电池注氦阀开
; rung 55
LD P_On
OUT TR0
LD 408.15  ; #3-2电池注氦阀开[M]
OR 608.15  ; #3-2电池注氦阀开[A]
ANDLD
SET 18.15  ; #3-2电池注氦阀开
LD TR0
LD 416.15  ; #3-2电池注氦阀关[M]
OR 616.15  ; #3-2电池注氦阀关[A]
ANDLD
RSET 18.15  ; #3-2电池注氦阀开

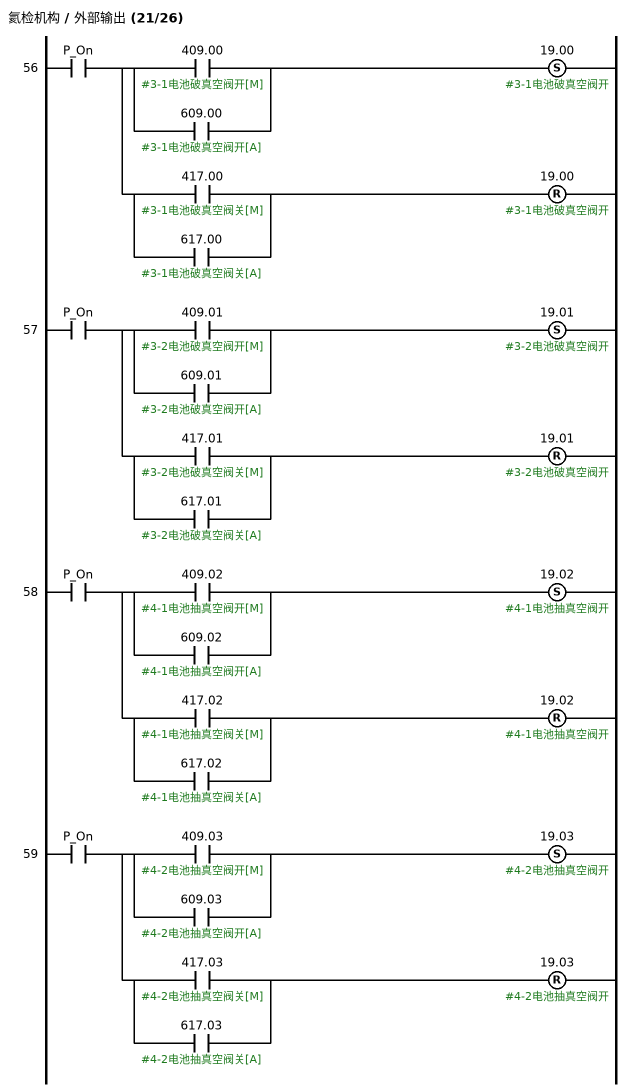
; rung 56
LD P_On
OUT TR0
LD 409.00  ; #3-1电池破真空阀开[M]
OR 609.00  ; #3-1电池破真空阀开[A]
ANDLD
SET 19.00  ; #3-1电池破真空阀开
LD TR0
LD 417.00  ; #3-1电池破真空阀关[M]
OR 617.00  ; #3-1电池破真空阀关[A]
ANDLD
RSET 19.00  ; #3-1电池破真空阀开
; rung 57
LD P_On
OUT TR0
LD 409.01  ; #3-2电池破真空阀开[M]
OR 609.01  ; #3-2电池破真空阀开[A]
ANDLD
SET 19.01  ; #3-2电池破真空阀开
LD TR0
LD 417.01  ; #3-2电池破真空阀关[M]
OR 617.01  ; #3-2电池破真空阀关[A]
ANDLD
RSET 19.01  ; #3-2电池破真空阀开
; rung 58
LD P_On
OUT TR0
LD 409.02  ; #4-1电池抽真空阀开[M]
OR 609.02  ; #4-1电池抽真空阀开[A]
ANDLD
SET 19.02  ; #4-1电池抽真空阀开
LD TR0
LD 417.02  ; #4-1电池抽真空阀关[M]
OR 617.02  ; #4-1电池抽真空阀关[A]
ANDLD
RSET 19.02  ; #4-1电池抽真空阀开
; rung 59
LD P_On
OUT TR0
LD 409.03  ; #4-2电池抽真空阀开[M]
OR 609.03  ; #4-2电池抽真空阀开[A]
ANDLD
SET 19.03  ; #4-2电池抽真空阀开
LD TR0
LD 417.03  ; #4-2电池抽真空阀关[M]
OR 617.03  ; #4-2电池抽真空阀关[A]
ANDLD
RSET 19.03  ; #4-2电池抽真空阀开

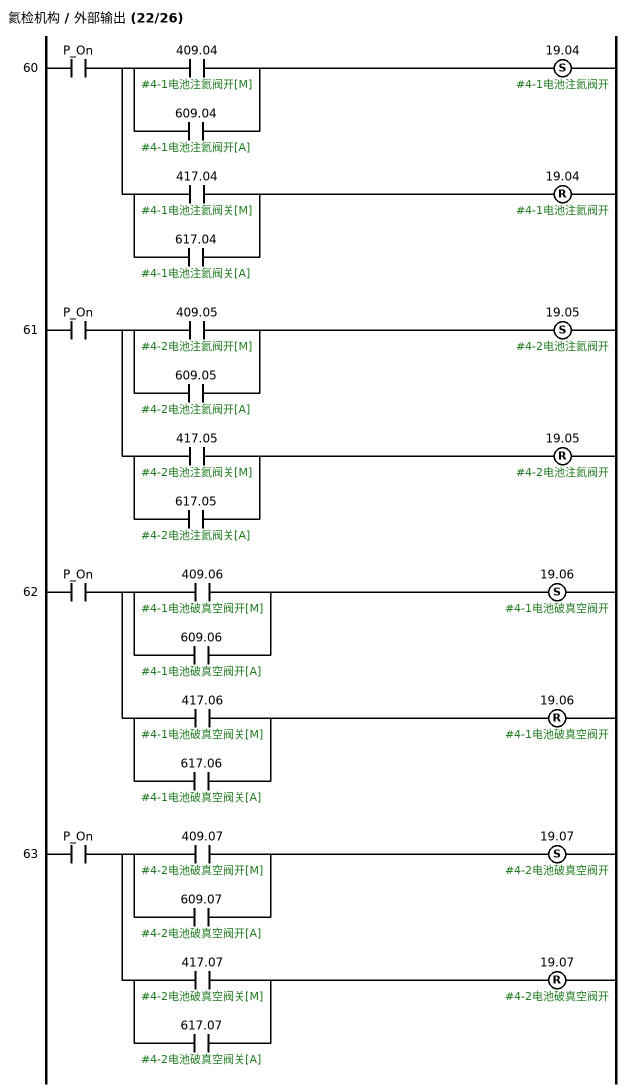
; rung 60
LD P_On
OUT TR0
LD 409.04  ; #4-1电池注氦阀开[M]
OR 609.04  ; #4-1电池注氦阀开[A]
ANDLD
SET 19.04  ; #4-1电池注氦阀开
LD TR0
LD 417.04  ; #4-1电池注氦阀关[M]
OR 617.04  ; #4-1电池注氦阀关[A]
ANDLD
RSET 19.04  ; #4-1电池注氦阀开
; rung 61
LD P_On
OUT TR0
LD 409.05  ; #4-2电池注氦阀开[M]
OR 609.05  ; #4-2电池注氦阀开[A]
ANDLD
SET 19.05  ; #4-2电池注氦阀开
LD TR0
LD 417.05  ; #4-2电池注氦阀关[M]
OR 617.05  ; #4-2电池注氦阀关[A]
ANDLD
RSET 19.05  ; #4-2电池注氦阀开
; rung 62
LD P_On
OUT TR0
LD 409.06  ; #4-1电池破真空阀开[M]
OR 609.06  ; #4-1电池破真空阀开[A]
ANDLD
SET 19.06  ; #4-1电池破真空阀开
LD TR0
LD 417.06  ; #4-1电池破真空阀关[M]
OR 617.06  ; #4-1电池破真空阀关[A]
ANDLD
RSET 19.06  ; #4-1电池破真空阀开
; rung 63
LD P_On
OUT TR0
LD 409.07  ; #4-2电池破真空阀开[M]
OR 609.07  ; #4-2电池破真空阀开[A]
ANDLD
SET 19.07  ; #4-2电池破真空阀开
LD TR0
LD 417.07  ; #4-2电池破真空阀关[M]
OR 617.07  ; #4-2电池破真空阀关[A]
ANDLD
RSET 19.07  ; #4-2电池破真空阀开

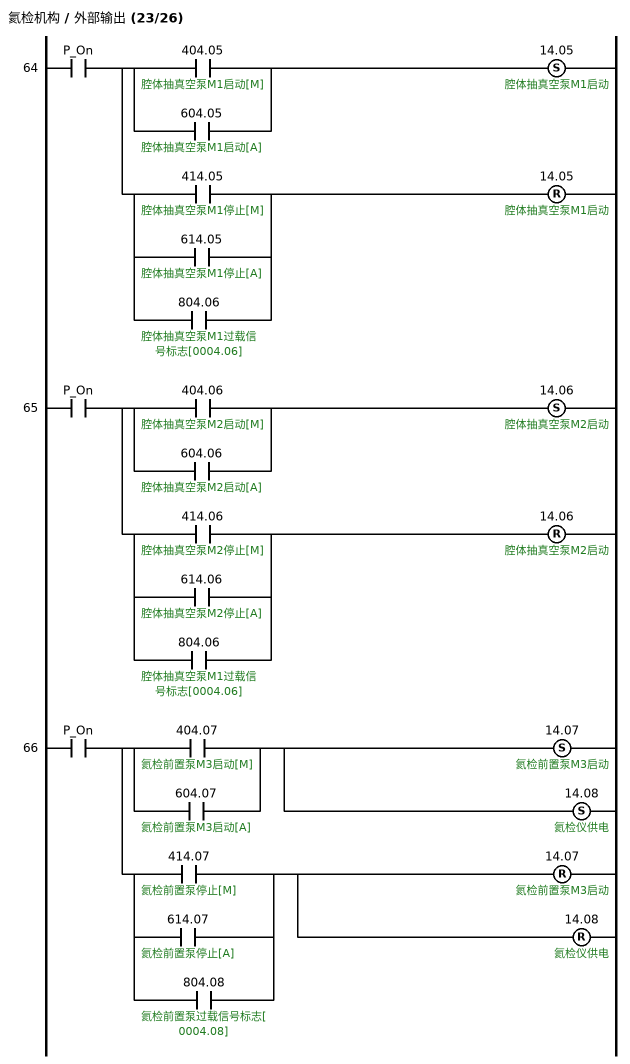
; rung 64
LD P_On
OUT TR0
LD 404.05  ; 腔体抽真空泵M1启动[M]
OR 604.05  ; 腔体抽真空泵M1启动[A]
ANDLD
SET 14.05  ; 腔体抽真空泵M1启动
LD TR0
LD 414.05  ; 腔体抽真空泵M1停止[M]
OR 614.05  ; 腔体抽真空泵M1停止[A]
OR 804.06  ; 腔体抽真空泵M1过载信号标志[0004.06]
ANDLD
RSET 14.05  ; 腔体抽真空泵M1启动
; rung 65
LD P_On
OUT TR0
LD 404.06  ; 腔体抽真空泵M2启动[M]
OR 604.06  ; 腔体抽真空泵M2启动[A]
ANDLD
SET 14.06  ; 腔体抽真空泵M2启动
LD TR0
LD 414.06  ; 腔体抽真空泵M2停止[M]
OR 614.06  ; 腔体抽真空泵M2停止[A]
OR 804.06  ; 腔体抽真空泵M1过载信号标志[0004.06]
ANDLD
RSET 14.06  ; 腔体抽真空泵M2启动
; rung 66
LD P_On
OUT TR0
LD 404.07  ; 氦检前置泵M3启动[M]
OR 604.07  ; 氦检前置泵M3启动[A]
ANDLD
SET 14.07  ; 氦检前置泵M3启动
SET 14.08  ; 氦检仪供电
LD TR0
LD 414.07  ; 氦检前置泵停止[M]
OR 614.07  ; 氦检前置泵停止[A]
OR 804.08  ; 氦检前置泵过载信号标志[0004.08]
ANDLD
RSET 14.07  ; 氦检前置泵M3启动
RSET 14.08  ; 氦检仪供电

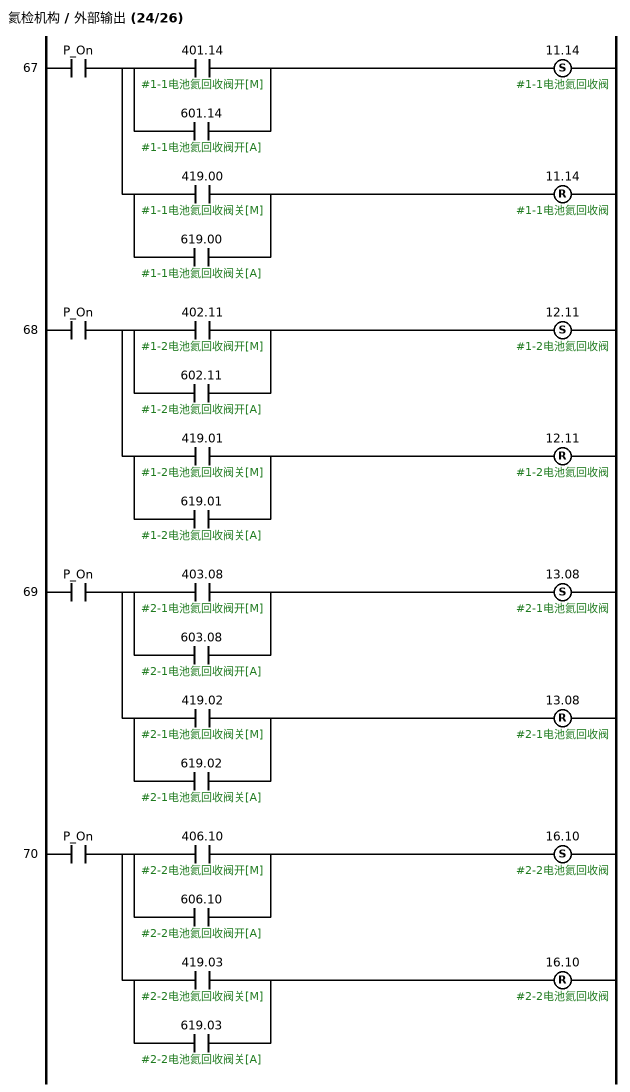
; rung 67
LD P_On
OUT TR0
LD 401.14  ; #1-1电池氦回收阀开[M]
OR 601.14  ; #1-1电池氦回收阀开[A]
ANDLD
SET 11.14  ; #1-1电池氦回收阀
LD TR0
LD 419.00  ; #1-1电池氦回收阀关[M]
OR 619.00  ; #1-1电池氦回收阀关[A]
ANDLD
RSET 11.14  ; #1-1电池氦回收阀
; rung 68
LD P_On
OUT TR0
LD 402.11  ; #1-2电池氦回收阀开[M]
OR 602.11  ; #1-2电池氦回收阀开[A]
ANDLD
SET 12.11  ; #1-2电池氦回收阀
LD TR0
LD 419.01  ; #1-2电池氦回收阀关[M]
OR 619.01  ; #1-2电池氦回收阀关[A]
ANDLD
RSET 12.11  ; #1-2电池氦回收阀
; rung 69
LD P_On
OUT TR0
LD 403.08  ; #2-1电池氦回收阀开[M]
OR 603.08  ; #2-1电池氦回收阀开[A]
ANDLD
SET 13.08  ; #2-1电池氦回收阀
LD TR0
LD 419.02  ; #2-1电池氦回收阀关[M]
OR 619.02  ; #2-1电池氦回收阀关[A]
ANDLD
RSET 13.08  ; #2-1电池氦回收阀
; rung 70
LD P_On
OUT TR0
LD 406.10  ; #2-2电池氦回收阀开[M]
OR 606.10  ; #2-2电池氦回收阀开[A]
ANDLD
SET 16.10  ; #2-2电池氦回收阀
LD TR0
LD 419.03  ; #2-2电池氦回收阀关[M]
OR 619.03  ; #2-2电池氦回收阀关[A]
ANDLD
RSET 16.10  ; #2-2电池氦回收阀

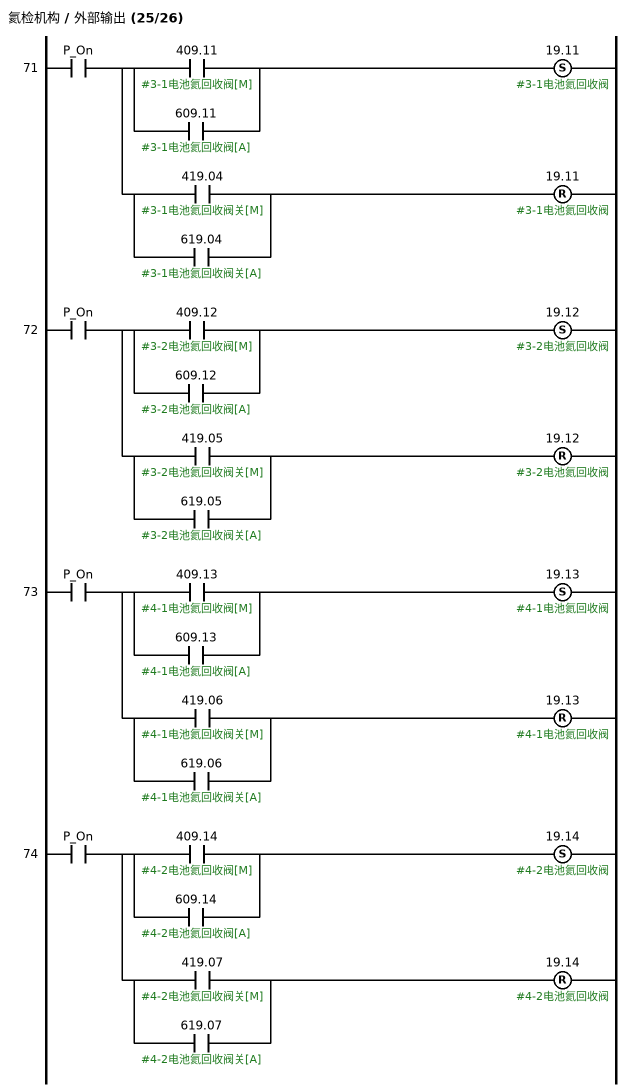
; rung 71
LD P_On
OUT TR0
LD 409.11  ; #3-1电池氦回收阀[M]
OR 609.11  ; #3-1电池氦回收阀[A]
ANDLD
SET 19.11  ; #3-1电池氦回收阀
LD TR0
LD 419.04  ; #3-1电池氦回收阀关[M]
OR 619.04  ; #3-1电池氦回收阀关[A]
ANDLD
RSET 19.11  ; #3-1电池氦回收阀
; rung 72
LD P_On
OUT TR0
LD 409.12  ; #3-2电池氦回收阀[M]
OR 609.12  ; #3-2电池氦回收阀[A]
ANDLD
SET 19.12  ; #3-2电池氦回收阀
LD TR0
LD 419.05  ; #3-2电池氦回收阀关[M]
OR 619.05  ; #3-2电池氦回收阀关[A]
ANDLD
RSET 19.12  ; #3-2电池氦回收阀
; rung 73
LD P_On
OUT TR0
LD 409.13  ; #4-1电池氦回收阀[M]
OR 609.13  ; #4-1电池氦回收阀[A]
ANDLD
SET 19.13  ; #4-1电池氦回收阀
LD TR0
LD 419.06  ; #4-1电池氦回收阀关[M]
OR 619.06  ; #4-1电池氦回收阀关[A]
ANDLD
RSET 19.13  ; #4-1电池氦回收阀
; rung 74
LD P_On
OUT TR0
LD 409.14  ; #4-2电池氦回收阀[M]
OR 609.14  ; #4-2电池氦回收阀[A]
ANDLD
SET 19.14  ; #4-2电池氦回收阀
LD TR0
LD 419.07  ; #4-2电池氦回收阀关[M]
OR 619.07  ; #4-2电池氦回收阀关[A]
ANDLD
RSET 19.14  ; #4-2电池氦回收阀

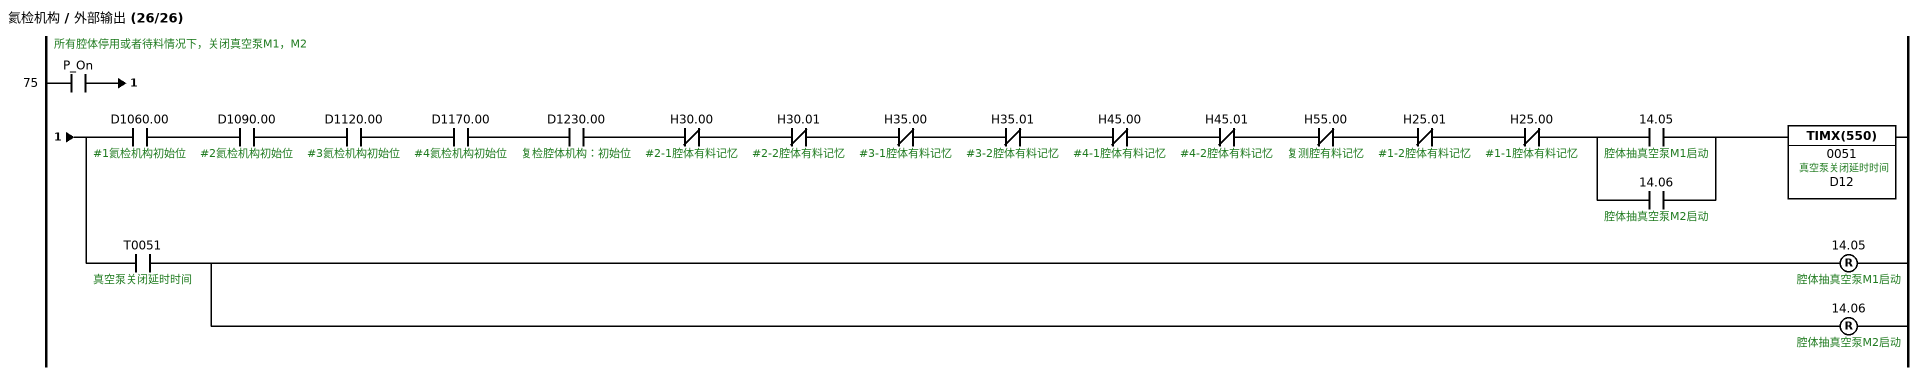
; rung 75: 所有腔体停用或者待料情况下，关闭真空泵M1，M2
LD P_On
OUT TR0
AND D1060.00  ; #1氦检机构初始位
AND D1090.00  ; #2氦检机构初始位
AND D1120.00  ; #3氦检机构初始位
AND D1170.00  ; #4氦检机构初始位
AND D1230.00  ; 复检腔体机构：初始位
ANDNOT H30.00  ; #2-1腔体有料记忆
ANDNOT H30.01  ; #2-2腔体有料记忆
ANDNOT H35.00  ; #3-1腔体有料记忆
ANDNOT H35.01  ; #3-2腔体有料记忆
ANDNOT H45.00  ; #4-1腔体有料记忆
ANDNOT H45.01  ; #4-2腔体有料记忆
ANDNOT H55.00  ; 复测腔有料记忆
ANDNOT H25.01  ; #1-2腔体有料记忆
ANDNOT H25.00  ; #1-1腔体有料记忆
LD 14.05  ; 腔体抽真空泵M1启动
OR 14.06  ; 腔体抽真空泵M2启动
ANDLD
TIMX(550) 0051 D12  ; 真空泵关闭延时时间
LD TR0
AND T0051  ; 真空泵关闭延时时间
RSET 14.05  ; 腔体抽真空泵M1启动
RSET 14.06  ; 腔体抽真空泵M2启动

### Section END
; rung 0
END(001)

## Program 出料伺服机构 (cyclic task 4)

### Section Main

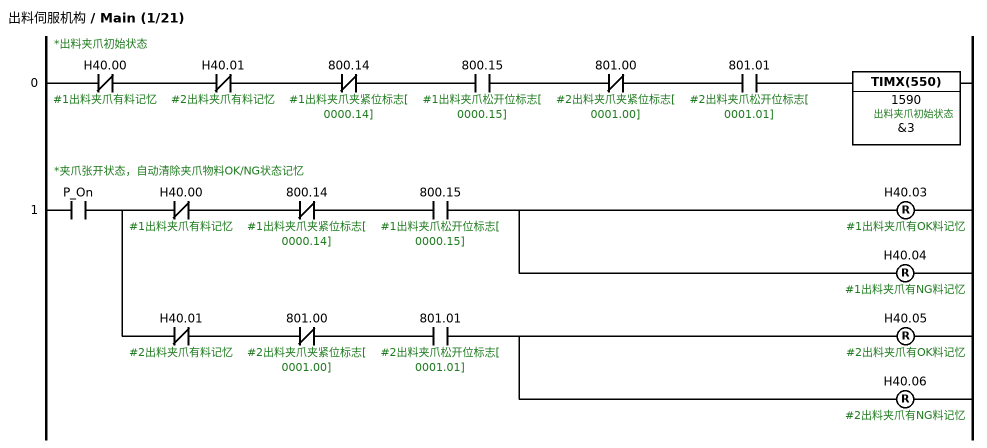
; rung 0: *出料夹爪初始状态
LDNOT H40.00  ; #1出料夹爪有料记忆
ANDNOT H40.01  ; #2出料夹爪有料记忆
ANDNOT 800.14  ; #1出料夹爪夹紧位标志[0000.14]
AND 800.15  ; #1出料夹爪松开位标志[0000.15]
ANDNOT 801.00  ; #2出料夹爪夹紧位标志[0001.00]
AND 801.01  ; #2出料夹爪松开位标志[0001.01]
TIMX(550) 1590 &3  ; 出料夹爪初始状态
; rung 1: *夹爪张开状态，自动清除夹爪物料OK/NG状态记忆
LD P_On
OUT TR0
ANDNOT H40.00  ; #1出料夹爪有料记忆
ANDNOT 800.14  ; #1出料夹爪夹紧位标志[0000.14]
AND 800.15  ; #1出料夹爪松开位标志[0000.15]
RSET H40.03  ; #1出料夹爪有OK料记忆
RSET H40.04  ; #1出料夹爪有NG料记忆
LD TR0
ANDNOT H40.01  ; #2出料夹爪有料记忆
ANDNOT 801.00  ; #2出料夹爪夹紧位标志[0001.00]
AND 801.01  ; #2出料夹爪松开位标志[0001.01]
RSET H40.05  ; #2出料夹爪有OK料记忆
RSET H40.06  ; #2出料夹爪有NG料记忆

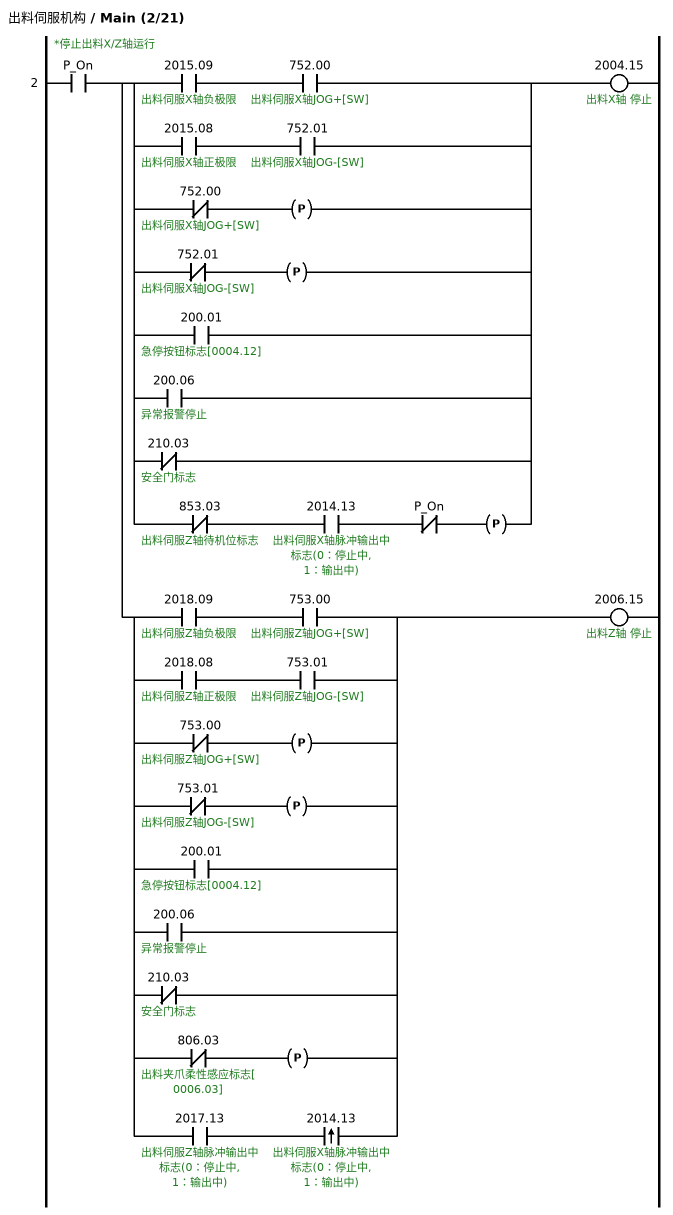
; rung 2: *停止出料X/Z轴运行
LD P_On
OUT TR0
LD 2015.09  ; 出料伺服X轴负极限
AND 752.00  ; 出料伺服X轴JOG+[SW]
LD 2015.08  ; 出料伺服X轴正极限
AND 752.01  ; 出料伺服X轴JOG-[SW]
ORLD
LDNOT 752.00  ; 出料伺服X轴JOG+[SW]
UP(521)
ORLD
LDNOT 752.01  ; 出料伺服X轴JOG-[SW]
UP(521)
ORLD
OR 200.01  ; 急停按钮标志[0004.12]
OR 200.06  ; 异常报警停止
ORNOT 210.03  ; 安全门标志
LDNOT 853.03  ; 出料伺服Z轴待机位标志
AND 2014.13  ; 出料伺服X轴脉冲输出中标志(0：停止中,1：输出中)
ANDNOT P_On
UP(521)
ORLD
ANDLD
OUT 2004.15  ; 出料X轴 停止
LD TR0
LD 2018.09  ; 出料伺服Z轴负极限
AND 753.00  ; 出料伺服Z轴JOG+[SW]
LD 2018.08  ; 出料伺服Z轴正极限
AND 753.01  ; 出料伺服Z轴JOG-[SW]
ORLD
LDNOT 753.00  ; 出料伺服Z轴JOG+[SW]
UP(521)
ORLD
LDNOT 753.01  ; 出料伺服Z轴JOG-[SW]
UP(521)
ORLD
OR 200.01  ; 急停按钮标志[0004.12]
OR 200.06  ; 异常报警停止
ORNOT 210.03  ; 安全门标志
LDNOT 806.03  ; 出料夹爪柔性感应标志[0006.03]
UP(521)
ORLD
LD 2017.13  ; 出料伺服Z轴脉冲输出中标志(0：停止中,1：输出中)
@AND 2014.13  ; 出料伺服X轴脉冲输出中标志(0：停止中,1：输出中)
ORLD
ANDLD
OUT 2006.15  ; 出料Z轴 停止

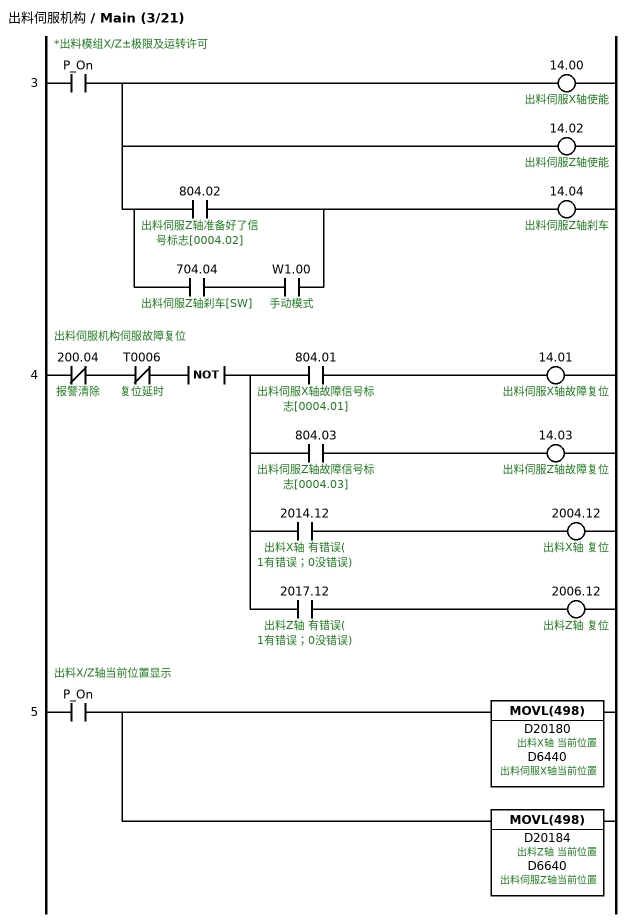
; rung 3: *出料模组X/Z±极限及运转许可
LD P_On
OUT 14.00  ; 出料伺服X轴使能
OUT 14.02  ; 出料伺服Z轴使能
LD 804.02  ; 出料伺服Z轴准备好了信号标志[0004.02]
LD 704.04  ; 出料伺服Z轴刹车[SW]
AND W1.00  ; 手动模式
ORLD
ANDLD
OUT 14.04  ; 出料伺服Z轴刹车
; rung 4: 出料伺服机构伺服故障复位
LDNOT 200.04  ; 报警清除
ANDNOT T0006  ; 复位延时
NOT(520)
OUT TR0
AND 804.01  ; 出料伺服X轴故障信号标志[0004.01]
OUT 14.01  ; 出料伺服X轴故障复位
LD TR0
AND 804.03  ; 出料伺服Z轴故障信号标志[0004.03]
OUT 14.03  ; 出料伺服Z轴故障复位
LD TR0
AND 2014.12  ; 出料X轴 有错误(1有错误；0没错误)
OUT 2004.12  ; 出料X轴 复位
LD TR0
AND 2017.12  ; 出料Z轴 有错误(1有错误；0没错误)
OUT 2006.12  ; 出料Z轴 复位
; rung 5: 出料X/Z轴当前位置显示
LD P_On
MOVL(498) D20180 D6440  ; 出料X轴 当前位置, 出料伺服X轴当前位置
MOVL(498) D20184 D6640  ; 出料Z轴 当前位置, 出料伺服Z轴当前位置

